C01816=1163.535,366.702,-80.590,-176.202,9.029,148.717
C01817=1163.539,366.455,-80.555,-176.204,9.026,148.716
C01818=1163.543,366.207,-80.520,-176.206,9.021,148.716
C01819=1163.547,365.925,-80.480,-176.209,9.017,148.716
C01820=1163.552,365.642,-80.440,-176.211,9.012,148.715
C01821=1163.557,365.360,-80.400,-176.214,9.008,148.715
C01822=1163.561,365.077,-80.360,-176.217,9.004,148.714
C01823=1163.565,364.830,-80.326,-176.219,9.000,148.714
C01824=1163.569,364.582,-80.290,-176.221,8.996,148.713
C01825=1163.573,364.334,-80.255,-176.223,8.993,148.713
C01826=1163.577,364.087,-80.220,-176.226,8.988,148.713
C01827=1163.581,363.840,-80.186,-176.228,8.985,148.712
C01828=1163.585,363.592,-80.152,-176.230,8.980,148.712
C01829=1163.589,363.345,-80.116,-176.233,8.977,148.712
C01830=1163.593,363.097,-80.081,-176.235,8.974,148.711
C01831=1163.597,362.849,-80.047,-176.237,8.969,148.711
C01832=1163.600,362.602,-80.012,-176.239,8.966,148.711
C01833=1163.605,362.355,-79.977,-176.242,8.962,148.710
C01834=1163.609,362.106,-79.942,-176.244,8.958,148.710
C01835=1163.612,361.860,-79.908,-176.247,8.954,148.710
C01836=1163.616,361.612,-79.873,-176.249,8.950,148.709
C01837=1163.621,361.364,-79.839,-176.252,8.946,148.709
C01838=1163.625,361.116,-79.804,-176.254,8.943,148.709
C01839=1163.628,360.870,-79.769,-176.256,8.939,148.708
C01840=1163.632,360.622,-79.734,-176.259,8.935,148.708
C01841=1163.637,360.374,-79.700,-176.261,8.932,148.708
C01842=1163.640,360.126,-79.666,-176.263,8.928,148.707
C01843=1163.645,359.879,-79.631,-176.265,8.924,148.707
C01844=1163.649,359.631,-79.596,-176.268,8.920,148.707
C01845=1163.652,359.384,-79.562,-176.270,8.917,148.706
C01846=1163.656,359.136,-79.527,-176.273,8.912,148.706
C01847=1163.661,358.889,-79.492,-176.275,8.909,148.706
C01848=1163.664,358.641,-79.458,-176.278,8.905,148.706
C01849=1163.669,358.394,-79.424,-176.280,8.901,148.705
C01850=1163.673,358.145,-79.389,-176.282,8.898,148.705
C01851=1163.676,357.898,-79.355,-176.285,8.894,148.705
C01852=1163.680,357.650,-79.320,-176.287,8.890,148.704
C01853=1163.684,357.403,-79.286,-176.290,8.886,148.704
C01854=1163.688,357.155,-79.251,-176.292,8.883,148.704
C01855=1163.692,356.908,-79.218,-176.294,8.880,148.704
C01856=1163.696,356.660,-79.183,-176.297,8.875,148.703
C01857=1163.701,356.412,-79.148,-176.299,8.872,148.703
C01858=1163.704,356.165,-79.114,-176.302,8.868,148.703
C01859=1163.708,355.917,-79.080,-176.304,8.864,148.702
C01860=1163.712,355.670,-79.046,-176.306,8.861,148.702
C01861=1163.716,355.422,-79.011,-176.309,8.857,148.702
C01862=1163.720,355.175,-78.977,-176.311,8.853,148.701
C01863=1163.725,354.927,-78.943,-176.314,8.849,148.701
C01864=1163.728,354.679,-78.909,-176.316,8.846,148.701
C01865=1163.733,354.432,-78.875,-176.318,8.842,148.701
C01866=1163.736,354.184,-78.840,-176.321,8.838,148.700
C01867=1163.740,353.936,-78.806,-176.324,8.835,148.700
C01868=1163.744,353.689,-78.772,-176.326,8.831,148.700
C01869=1163.748,353.441,-78.737,-176.328,8.827,148.699
C01870=1163.752,353.193,-78.704,-176.331,8.824,148.699
C01871=1163.756,352.946,-78.670,-176.334,8.820,148.699
C01872=1163.760,352.698,-78.635,-176.335,8.816,148.698
C01873=1163.764,352.451,-78.601,-176.338,8.813,148.698
C01874=1163.769,352.203,-78.568,-176.341,8.809,148.698
C01875=1163.772,351.955,-78.533,-176.343,8.806,148.698
C01876=1163.777,351.708,-78.499,-176.346,8.801,148.698
C01877=1163.781,351.460,-78.466,-176.348,8.798,148.697
C01878=1163.784,351.212,-78.432,-176.350,8.795,148.697
C01879=1163.789,350.965,-78.397,-176.353,8.790,148.697
C01880=1163.793,350.717,-78.364,-176.355,8.787,148.696
C01881=1163.796,350.469,-78.330,-176.357,8.784,148.696
C01882=1163.801,350.222,-78.295,-176.360,8.780,148.696
C01883=1163.805,349.974,-78.262,-176.363,8.776,148.696
C01884=1163.809,349.727,-78.228,-176.365,8.773,148.696
C01885=1163.813,349.478,-78.194,-176.367,8.769,148.695
C01886=1163.817,349.231,-78.160,-176.370,8.765,148.695
C01887=1163.821,348.983,-78.127,-176.372,8.762,148.695
C01888=1163.825,348.736,-78.093,-176.375,8.758,148.694
C01889=1163.829,348.488,-78.059,-176.377,8.755,148.694
C01890=1163.833,348.240,-78.025,-176.379,8.752,148.694
C01891=1163.837,347.993,-77.992,-176.382,8.747,148.694
C01892=1163.841,347.745,-77.958,-176.384,8.744,148.693
C01893=1163.845,347.497,-77.924,-176.387,8.741,148.693
C01894=1163.849,347.250,-77.890,-176.389,8.736,148.693
C01895=1163.853,347.002,-77.857,-176.391,8.733,148.693
C01896=1163.858,346.755,-77.823,-176.394,8.730,148.692
C01897=1163.862,346.507,-77.789,-176.397,8.726,148.692
C01898=1163.865,346.258,-77.756,-176.399,8.722,148.692
C01899=1163.869,346.011,-77.722,-176.401,8.719,148.692
C01900=1163.873,345.764,-77.689,-176.404,8.715,148.691
C01901=1163.878,345.516,-77.655,-176.406,8.712,148.691
C01902=1163.882,345.268,-77.621,-176.409,8.708,148.691
C01903=1163.885,345.020,-77.588,-176.412,8.704,148.691
C01904=1163.890,344.772,-77.555,-176.414,8.701,148.691
C01905=1163.893,344.525,-77.521,-176.416,8.698,148.690
C01906=1163.898,344.277,-77.488,-176.419,8.694,148.690
C01907=1163.902,344.029,-77.454,-176.421,8.690,148.690
C01908=1163.907,343.782,-77.421,-176.424,8.687,148.690
C01909=1163.910,343.534,-77.386,-176.426,8.684,148.689
C01910=1163.914,343.286,-77.353,-176.429,8.680,148.689
C01911=1163.918,343.038,-77.320,-176.431,8.676,148.689
C01912=1163.922,342.791,-77.287,-176.433,8.673,148.689
C01913=1163.926,342.543,-77.254,-176.436,8.669,148.688
C01914=1163.930,342.296,-77.220,-176.439,8.666,148.688
C01915=1163.934,342.048,-77.187,-176.441,8.662,148.688
C01916=1163.938,341.800,-77.154,-176.444,8.658,148.688
C01917=1163.943,341.553,-77.120,-176.446,8.655,148.688
C01918=1163.947,341.304,-77.086,-176.448,8.652,148.687
C01919=1163.951,341.056,-77.053,-176.451,8.648,148.687
C01920=1163.955,340.808,-77.020,-176.454,8.644,148.687
C01921=1163.959,340.561,-76.987,-176.456,8.641,148.687
C01922=1163.963,340.313,-76.954,-176.458,8.638,148.687
C01923=1163.968,340.033,-76.916,-176.461,8.634,148.686
C01924=1163.973,339.754,-76.879,-176.464,8.629,148.686
C01925=1163.977,339.474,-76.841,-176.467,8.625,148.686
C01926=1163.981,339.195,-76.804,-176.470,8.621,148.686
C01927=1163.985,338.947,-76.771,-176.472,8.618,148.685
C01928=1163.989,338.700,-76.738,-176.474,8.615,148.685
C01929=1163.993,338.452,-76.705,-176.477,8.612,148.685
C01930=1163.998,338.204,-76.672,-176.480,8.608,148.685
C01931=1164.002,337.956,-76.638,-176.482,8.604,148.685
C01932=1164.006,337.709,-76.605,-176.484,8.601,148.684
C01933=1164.010,337.461,-76.572,-176.487,8.598,148.684
C01934=1164.014,337.213,-76.540,-176.490,8.594,148.684
C01935=1164.019,336.965,-76.507,-176.492,8.590,148.684
C01936=1164.022,336.717,-76.474,-176.494,8.587,148.684
C01937=1164.026,336.470,-76.441,-176.496,8.584,148.683
C01938=1164.030,336.222,-76.408,-176.499,8.580,148.683
C01939=1164.034,335.974,-76.374,-176.502,8.577,148.683
C01940=1164.039,335.726,-76.342,-176.504,8.573,148.683
C01941=1164.043,335.478,-76.309,-176.507,8.570,148.683
C01942=1164.046,335.231,-76.276,-176.510,8.566,148.682
C01943=1164.051,334.983,-76.243,-176.512,8.563,148.682
C01944=1164.055,334.735,-76.211,-176.514,8.559,148.682
C01945=1164.059,334.487,-76.178,-176.516,8.556,148.682
C01946=1164.063,334.239,-76.144,-176.520,8.552,148.682
C01947=1164.067,333.991,-76.113,-176.522,8.549,148.682
C01948=1164.071,333.743,-76.079,-176.524,8.546,148.681
C01949=1164.075,333.496,-76.046,-176.527,8.542,148.681
C01950=1164.080,333.247,-76.014,-176.529,8.538,148.681
C01951=1164.083,333.000,-75.981,-176.532,8.535,148.681
C01952=1164.088,332.753,-75.948,-176.535,8.532,148.681
C01953=1164.092,332.505,-75.916,-176.537,8.529,148.681
C01954=1164.096,332.257,-75.883,-176.539,8.525,148.680
C01955=1164.100,332.009,-75.850,-176.542,8.521,148.680
C01956=1164.104,331.761,-75.818,-176.544,8.518,148.680
C01957=1164.108,331.513,-75.785,-176.547,8.515,148.680
C01958=1164.112,331.265,-75.753,-176.549,8.512,148.680
C01959=1164.116,331.018,-75.720,-176.552,8.508,148.679
C01960=1164.121,330.769,-75.687,-176.554,8.504,148.679
C01961=1164.125,330.522,-75.655,-176.557,8.501,148.679
C01962=1164.129,330.274,-75.623,-176.559,8.498,148.679
C01963=1164.133,330.026,-75.589,-176.562,8.495,148.679
C01964=1164.137,329.778,-75.558,-176.565,8.491,148.679
C01965=1164.141,329.531,-75.524,-176.567,8.487,148.678
C01966=1164.145,329.283,-75.493,-176.569,8.484,148.678
C01967=1164.149,329.034,-75.460,-176.572,8.481,148.678
C01968=1164.154,328.787,-75.427,-176.574,8.478,148.678
C01969=1164.158,328.539,-75.396,-176.577,8.474,148.678
C01970=1164.162,328.291,-75.362,-176.579,8.470,148.678
C01971=1164.166,328.043,-75.331,-176.582,8.467,148.678
C01972=1164.170,327.795,-75.298,-176.584,8.464,148.677
C01973=1164.174,327.548,-75.266,-176.587,8.461,148.677
C01974=1164.178,327.300,-75.233,-176.590,8.457,148.677
C01975=1164.182,327.052,-75.202,-176.592,8.454,148.677
C01976=1164.186,326.804,-75.168,-176.595,8.451,148.677
C01977=1164.190,326.556,-75.137,-176.597,8.447,148.677
C01978=1164.195,326.309,-75.105,-176.599,8.444,148.676
C01979=1164.199,326.060,-75.073,-176.603,8.440,148.676
C01980=1164.203,325.813,-75.040,-176.605,8.437,148.676
C01981=1164.207,325.565,-75.008,-176.607,8.434,148.676
C01982=1164.211,325.316,-74.975,-176.609,8.430,148.676
C01983=1164.215,325.069,-74.944,-176.612,8.427,148.676
C01984=1164.220,324.821,-74.911,-176.615,8.423,148.675
C01985=1164.223,324.573,-74.879,-176.617,8.420,148.675
C01986=1164.228,324.325,-74.846,-176.620,8.417,148.675
C01987=1164.232,324.078,-74.815,-176.622,8.414,148.675
C01988=1164.236,323.830,-74.783,-176.625,8.410,148.675
C01989=1164.240,323.581,-74.751,-176.627,8.407,148.675
C01990=1164.244,323.333,-74.719,-176.630,8.403,148.675
C01991=1164.249,323.085,-74.687,-176.633,8.400,148.674
C01992=1164.253,322.837,-74.655,-176.635,8.397,148.674
C01993=1164.256,322.589,-74.623,-176.638,8.394,148.674
C01994=1164.261,322.342,-74.591,-176.640,8.390,148.674
C01995=1164.265,322.094,-74.559,-176.642,8.387,148.674
C01996=1164.268,321.846,-74.526,-176.646,8.383,148.674
C01997=1164.273,321.599,-74.494,-176.648,8.380,148.674
C01998=1164.277,321.351,-74.463,-176.650,8.377,148.673
C01999=1164.281,321.102,-74.431,-176.653,8.374,148.673
C02000=1164.286,320.854,-74.399,-176.655,8.370,148.673
C02001=1164.290,320.606,-74.368,-176.657,8.367,148.673
C02002=1164.294,320.358,-74.336,-176.661,8.363,148.673
C02003=1164.298,320.111,-74.304,-176.663,8.360,148.673
C02004=1164.302,319.863,-74.272,-176.665,8.357,148.673
C02005=1164.306,319.615,-74.240,-176.668,8.354,148.673
C02006=1164.310,319.367,-74.208,-176.670,8.351,148.672
C02007=1164.314,319.119,-74.177,-176.673,8.348,148.672
C02008=1164.319,318.871,-74.144,-176.675,8.344,148.672
C02009=1164.323,318.623,-74.113,-176.678,8.340,148.672
C02010=1164.327,318.375,-74.082,-176.681,8.337,148.672
C02011=1164.331,318.127,-74.050,-176.683,8.334,148.672
C02012=1164.336,317.879,-74.018,-176.686,8.331,148.672
C02013=1164.339,317.631,-73.986,-176.688,8.328,148.672
C02014=1164.344,317.383,-73.955,-176.691,8.324,148.671
C02015=1164.348,317.135,-73.923,-176.693,8.321,148.672
C02016=1164.351,316.887,-73.891,-176.696,8.317,148.671
C02017=1164.356,316.640,-73.860,-176.699,8.314,148.671
C02018=1164.360,316.391,-73.828,-176.701,8.311,148.671
C02019=1164.365,316.143,-73.797,-176.704,8.308,148.671
C02020=1164.368,315.895,-73.765,-176.706,8.305,148.671
C02021=1164.373,315.647,-73.734,-176.709,8.301,148.671
C02022=1164.377,315.399,-73.702,-176.711,8.298,148.671
C02023=1164.380,315.151,-73.670,-176.714,8.295,148.671
C02024=1164.385,314.903,-73.640,-176.717,8.291,148.670
C02025=1164.389,314.655,-73.608,-176.719,8.288,148.670
C02026=1164.393,314.408,-73.576,-176.722,8.285,148.670
C02027=1164.398,314.131,-73.542,-176.724,8.282,148.670
C02028=1164.403,313.853,-73.506,-176.727,8.278,148.670
C02029=1164.407,313.576,-73.471,-176.731,8.274,148.670
C02030=1164.412,313.299,-73.436,-176.733,8.271,148.670
C02031=1164.416,313.051,-73.405,-176.736,8.268,148.670
C02032=1164.421,312.803,-73.373,-176.738,8.264,148.670
C02033=1164.425,312.555,-73.342,-176.741,8.260,148.669
C02034=1164.429,312.307,-73.310,-176.744,8.257,148.669
C02035=1164.433,312.059,-73.279,-176.746,8.254,148.669
C02036=1164.437,311.811,-73.248,-176.749,8.251,148.669
C02037=1164.441,311.563,-73.217,-176.751,8.248,148.669
C02038=1164.446,311.315,-73.185,-176.754,8.245,148.669
C02039=1164.450,311.067,-73.154,-176.756,8.241,148.669
C02040=1164.454,310.819,-73.123,-176.759,8.239,148.669
C02041=1164.458,310.571,-73.091,-176.761,8.235,148.669
C02042=1164.463,310.323,-73.061,-176.764,8.231,148.669
C02043=1164.467,310.075,-73.030,-176.767,8.228,148.668
C02044=1164.470,309.827,-72.999,-176.769,8.225,148.668
C02045=1164.475,309.579,-72.968,-176.772,8.222,148.668
C02046=1164.479,309.330,-72.937,-176.774,8.219,148.668
C02047=1164.483,309.083,-72.905,-176.777,8.216,148.668
C02048=1164.487,308.834,-72.874,-176.779,8.213,148.668
C02049=1164.492,308.587,-72.843,-176.782,8.209,148.668
C02050=1164.496,308.339,-72.812,-176.784,8.206,148.668
C02051=1164.500,308.091,-72.781,-176.787,8.203,148.668
C02052=1164.505,307.843,-72.750,-176.789,8.200,148.668
C02053=1164.508,307.594,-72.720,-176.792,8.196,148.668
C02054=1164.512,307.347,-72.688,-176.795,8.193,148.668
C02055=1164.517,307.099,-72.657,-176.797,8.190,148.667
C02056=1164.521,306.850,-72.626,-176.800,8.187,148.667
C02057=1164.526,306.602,-72.595,-176.802,8.184,148.667
C02058=1164.530,306.354,-72.565,-176.805,8.181,148.667
C02059=1164.533,306.106,-72.534,-176.807,8.177,148.667
C02060=1164.538,305.859,-72.503,-176.810,8.174,148.667
C02061=1164.542,305.611,-72.472,-176.812,8.171,148.667
C02062=1164.546,305.362,-72.441,-176.815,8.168,148.667
C02063=1164.551,305.114,-72.410,-176.818,8.165,148.667
C02064=1164.555,304.866,-72.380,-176.820,8.162,148.667
C02065=1164.559,304.618,-72.349,-176.823,8.158,148.667
C02066=1164.563,304.370,-72.318,-176.825,8.155,148.667
C02067=1164.568,304.122,-72.287,-176.828,8.151,148.666
C02068=1164.571,303.874,-72.257,-176.831,8.148,148.666
C02069=1164.576,303.626,-72.226,-176.834,8.145,148.666
C02070=1164.581,303.378,-72.195,-176.836,8.142,148.666
C02071=1164.584,303.130,-72.165,-176.839,8.139,148.666
C02072=1164.588,302.881,-72.134,-176.841,8.136,148.666
C02073=1164.593,302.633,-72.103,-176.844,8.133,148.666
C02074=1164.597,302.386,-72.073,-176.846,8.130,148.666
C02075=1164.601,302.137,-72.042,-176.849,8.127,148.666
C02076=1164.606,301.889,-72.011,-176.852,8.124,148.666
C02077=1164.609,301.641,-71.981,-176.854,8.120,148.666
C02078=1164.614,301.393,-71.950,-176.857,8.117,148.666
C02079=1164.618,301.144,-71.920,-176.859,8.114,148.666
C02080=1164.622,300.897,-71.889,-176.862,8.111,148.666
C02081=1164.627,300.649,-71.859,-176.864,8.108,148.665
C02082=1164.631,300.401,-71.828,-176.867,8.105,148.665
C02083=1164.635,300.153,-71.798,-176.869,8.102,148.666
C02084=1164.639,299.904,-71.767,-176.872,8.099,148.665
C02085=1164.644,299.656,-71.737,-176.874,8.096,148.665
C02086=1164.648,299.408,-71.706,-176.877,8.092,148.665
C02087=1164.652,299.160,-71.676,-176.880,8.089,148.665
C02088=1164.656,298.912,-71.645,-176.883,8.086,148.665
C02089=1164.660,298.664,-71.616,-176.885,8.082,148.665
C02090=1164.665,298.416,-71.585,-176.888,8.079,148.665
C02091=1164.669,298.168,-71.555,-176.891,8.076,148.665
C02092=1164.673,297.920,-71.524,-176.893,8.073,148.665
C02093=1164.678,297.672,-71.494,-176.896,8.070,148.665
C02094=1164.682,297.423,-71.463,-176.898,8.067,148.665
C02095=1164.685,297.175,-71.433,-176.901,8.064,148.665
C02096=1164.690,296.927,-71.403,-176.903,8.061,148.665
C02097=1164.694,296.679,-71.373,-176.906,8.058,148.665
C02098=1164.699,296.431,-71.343,-176.908,8.055,148.665
C02099=1164.703,296.183,-71.313,-176.911,8.052,148.665
C02100=1164.707,295.934,-71.282,-176.914,8.048,148.665
C02101=1164.711,295.686,-71.252,-176.916,8.045,148.665
C02102=1164.716,295.438,-71.221,-176.919,8.042,148.664
C02103=1164.720,295.190,-71.192,-176.921,8.039,148.664
C02104=1164.724,294.942,-71.162,-176.924,8.036,148.664
C02105=1164.729,294.694,-71.132,-176.926,8.033,148.664
C02106=1164.733,294.446,-71.102,-176.929,8.030,148.664
C02107=1164.737,294.198,-71.072,-176.932,8.027,148.664
C02108=1164.741,293.949,-71.041,-176.934,8.024,148.664
C02109=1164.745,293.701,-71.012,-176.937,8.021,148.664
C02110=1164.750,293.453,-70.981,-176.940,8.018,148.664
C02111=1164.754,293.204,-70.951,-176.942,8.015,148.664
C02112=1164.758,292.957,-70.921,-176.945,8.012,148.664
C02113=1164.763,292.708,-70.891,-176.947,8.009,148.664
C02114=1164.766,292.461,-70.861,-176.950,8.006,148.664
C02115=1164.771,292.212,-70.831,-176.952,8.002,148.664
C02116=1164.775,291.964,-70.802,-176.955,7.999,148.664
C02117=1164.779,291.716,-70.771,-176.958,7.996,148.664
C02118=1164.784,291.468,-70.742,-176.960,7.993,148.664
C02119=1164.788,291.220,-70.712,-176.963,7.990,148.664
C02120=1164.792,290.972,-70.682,-176.966,7.987,148.664
C02121=1164.797,290.723,-70.652,-176.968,7.984,148.664
C02122=1164.801,290.475,-70.623,-176.971,7.981,148.664
C02123=1164.805,290.227,-70.592,-176.974,7.978,148.664
C02124=1164.810,289.979,-70.562,-176.976,7.975,148.664
C02125=1164.813,289.730,-70.533,-176.979,7.972,148.664
C02126=1164.817,289.482,-70.503,-176.981,7.969,148.664
C02127=1164.821,289.234,-70.473,-176.984,7.966,148.664
C02128=1164.825,288.986,-70.444,-176.986,7.962,148.664
C02129=1164.831,288.738,-70.414,-176.989,7.960,148.664
C02130=1164.835,288.490,-70.384,-176.992,7.957,148.664
C02131=1164.840,288.215,-70.351,-176.995,7.954,148.664
C02132=1164.844,287.940,-70.319,-176.998,7.949,148.663
C02133=1164.849,287.665,-70.286,-177.000,7.947,148.663
C02134=1164.854,287.390,-70.253,-177.004,7.943,148.663
C02135=1164.858,287.141,-70.224,-177.006,7.940,148.663
C02136=1164.862,286.893,-70.194,-177.009,7.938,148.664
C02137=1164.867,286.645,-70.163,-177.011,7.934,148.663
C02138=1164.871,286.397,-70.134,-177.014,7.931,148.663
C02139=1164.875,286.149,-70.105,-177.016,7.928,148.663
C02140=1164.879,285.900,-70.075,-177.019,7.925,148.664
C02141=1164.883,285.652,-70.046,-177.021,7.922,148.663
C02142=1164.887,285.404,-70.016,-177.024,7.919,148.663
C02143=1164.892,285.155,-69.987,-177.027,7.916,148.663
C02144=1164.896,284.908,-69.958,-177.030,7.913,148.663
C02145=1164.901,284.660,-69.928,-177.032,7.910,148.663
C02146=1164.905,284.411,-69.899,-177.035,7.907,148.663
C02147=1164.909,284.163,-69.869,-177.037,7.904,148.663
C02148=1164.913,283.915,-69.840,-177.040,7.901,148.663
C02149=1164.917,283.667,-69.810,-177.042,7.898,148.663
C02150=1164.922,283.418,-69.782,-177.045,7.895,148.663
C02151=1164.926,283.169,-69.752,-177.048,7.892,148.663
C02152=1164.931,282.922,-69.723,-177.051,7.889,148.663
C02153=1164.935,282.674,-69.694,-177.053,7.886,148.663
C02154=1164.939,282.425,-69.664,-177.056,7.883,148.663
C02155=1164.943,282.177,-69.635,-177.059,7.880,148.663
C02156=1164.947,281.929,-69.605,-177.061,7.877,148.663
C02157=1164.952,281.680,-69.577,-177.064,7.874,148.663
C02158=1164.956,281.432,-69.547,-177.066,7.872,148.663
C02159=1164.961,281.184,-69.518,-177.068,7.868,148.663
C02160=1164.965,280.936,-69.489,-177.071,7.865,148.663
C02161=1164.969,280.688,-69.459,-177.074,7.862,148.663
C02162=1164.974,280.439,-69.430,-177.077,7.859,148.663
C02163=1164.978,280.190,-69.401,-177.079,7.856,148.663
C02164=1164.983,279.943,-69.372,-177.082,7.853,148.663
C02165=1164.987,279.695,-69.342,-177.085,7.850,148.663
C02166=1164.991,279.446,-69.314,-177.087,7.847,148.663
C02167=1164.995,279.198,-69.285,-177.090,7.844,148.663
C02168=1164.999,278.949,-69.255,-177.093,7.841,148.663
C02169=1165.004,278.701,-69.227,-177.096,7.838,148.663
C02170=1165.008,278.453,-69.198,-177.098,7.835,148.663
C02171=1165.013,278.205,-69.168,-177.101,7.832,148.663
C02172=1165.016,277.956,-69.140,-177.103,7.829,148.663
C02173=1165.021,277.709,-69.111,-177.106,7.827,148.663
C02174=1165.026,277.460,-69.082,-177.108,7.824,148.664
C02175=1165.030,277.211,-69.053,-177.111,7.821,148.664
C02176=1165.034,276.963,-69.023,-177.114,7.818,148.664
C02177=1165.038,276.715,-68.995,-177.116,7.815,148.663
C02178=1165.042,276.467,-68.966,-177.119,7.812,148.663
C02179=1165.047,276.218,-68.937,-177.122,7.809,148.664
C02180=1165.051,275.970,-68.908,-177.124,7.806,148.664
C02181=1165.055,275.722,-68.880,-177.127,7.803,148.664
C02182=1165.060,275.474,-68.851,-177.130,7.800,148.664
C02183=1165.064,275.225,-68.822,-177.133,7.797,148.664
C02184=1165.068,274.977,-68.793,-177.134,7.795,148.664
C02185=1165.073,274.729,-68.765,-177.137,7.792,148.664
C02186=1165.077,274.480,-68.735,-177.140,7.789,148.664
C02187=1165.081,274.232,-68.706,-177.143,7.786,148.664
C02188=1165.086,273.984,-68.679,-177.145,7.783,148.664
C02189=1165.090,273.735,-68.649,-177.148,7.780,148.664
C02190=1165.094,273.486,-68.620,-177.151,7.777,148.664
C02191=1165.099,273.239,-68.593,-177.154,7.774,148.664
C02192=1165.103,272.990,-68.563,-177.156,7.771,148.664
C02193=1165.107,272.742,-68.535,-177.158,7.768,148.664
C02194=1165.111,272.494,-68.506,-177.161,7.765,148.664
C02195=1165.116,272.245,-68.477,-177.164,7.763,148.664
C02196=1165.120,271.997,-68.449,-177.166,7.760,148.664
C02197=1165.125,271.749,-68.421,-177.169,7.757,148.664
C02198=1165.129,271.500,-68.391,-177.172,7.754,148.664
C02199=1165.133,271.252,-68.363,-177.175,7.751,148.664
C02200=1165.138,271.004,-68.335,-177.177,7.748,148.664
C02201=1165.141,270.755,-68.307,-177.180,7.745,148.664
C02202=1165.146,270.507,-68.278,-177.182,7.743,148.664
C02203=1165.150,270.259,-68.249,-177.185,7.740,148.664
C02204=1165.155,270.011,-68.221,-177.188,7.737,148.664
C02205=1165.159,269.762,-68.193,-177.190,7.733,148.664
C02206=1165.163,269.513,-68.164,-177.193,7.730,148.664
C02207=1165.168,269.266,-68.135,-177.196,7.728,148.664
C02208=1165.172,269.017,-68.107,-177.198,7.725,148.664
C02209=1165.177,268.769,-68.079,-177.201,7.722,148.664
C02210=1165.181,268.520,-68.050,-177.203,7.719,148.665
C02211=1165.186,268.272,-68.022,-177.206,7.716,148.665
C02212=1165.190,268.023,-67.994,-177.209,7.714,148.665
C02213=1165.194,267.776,-67.966,-177.212,7.711,148.665
C02214=1165.198,267.527,-67.937,-177.214,7.708,148.665
C02215=1165.202,267.278,-67.909,-177.217,7.705,148.665
C02216=1165.207,267.030,-67.881,-177.220,7.702,148.665
C02217=1165.211,266.781,-67.853,-177.222,7.700,148.665
C02218=1165.216,266.533,-67.824,-177.225,7.697,148.665
C02219=1165.220,266.285,-67.796,-177.228,7.694,148.665
C02220=1165.225,266.036,-67.768,-177.230,7.691,148.665
C02221=1165.229,265.788,-67.740,-177.233,7.688,148.665
C02222=1165.233,265.540,-67.712,-177.236,7.685,148.665
C02223=1165.237,265.291,-67.683,-177.238,7.683,148.665
C02224=1165.242,265.043,-67.655,-177.241,7.680,148.665
C02225=1165.246,264.794,-67.627,-177.243,7.677,148.665
C02226=1165.251,264.546,-67.599,-177.246,7.674,148.665
C02227=1165.254,264.298,-67.571,-177.249,7.671,148.666
C02228=1165.260,264.050,-67.542,-177.252,7.668,148.666
C02229=1165.264,263.802,-67.515,-177.255,7.665,148.666
C02230=1165.268,263.553,-67.486,-177.257,7.663,148.666
C02231=1165.273,263.304,-67.459,-177.259,7.660,148.666
C02232=1165.277,263.056,-67.431,-177.262,7.657,148.666
C02233=1165.281,262.808,-67.403,-177.265,7.654,148.666
C02234=1165.285,262.559,-67.375,-177.268,7.651,148.666
C02235=1165.290,262.286,-67.343,-177.270,7.648,148.666
C02236=1165.296,262.013,-67.313,-177.273,7.645,148.666
C02237=1165.300,261.740,-67.282,-177.276,7.642,148.666
C02238=1165.305,261.466,-67.252,-177.279,7.638,148.666
C02239=1165.309,261.219,-67.224,-177.282,7.636,148.666
C02240=1165.313,260.970,-67.196,-177.284,7.633,148.666
C02241=1165.318,260.722,-67.169,-177.287,7.630,148.666
C02242=1165.322,260.473,-67.140,-177.290,7.627,148.666
C02243=1165.326,260.225,-67.112,-177.293,7.624,148.666
C02244=1165.331,259.976,-67.085,-177.295,7.622,148.667
C02245=1165.335,259.728,-67.057,-177.297,7.619,148.667
C02246=1165.339,259.480,-67.029,-177.300,7.616,148.667
C02247=1165.345,259.231,-67.002,-177.303,7.613,148.667
C02248=1165.348,258.982,-66.973,-177.306,7.611,148.667
C02249=1165.353,258.735,-66.946,-177.308,7.609,148.667
C02250=1165.357,258.485,-66.918,-177.311,7.606,148.667
C02251=1165.361,258.237,-66.890,-177.314,7.603,148.667
C02252=1165.366,257.989,-66.863,-177.317,7.600,148.667
C02253=1165.370,257.740,-66.835,-177.319,7.597,148.667
C02254=1165.375,257.492,-66.808,-177.322,7.595,148.667
C02255=1165.379,257.244,-66.780,-177.324,7.592,148.667
C02256=1165.383,256.995,-66.752,-177.327,7.589,148.668
C02257=1165.388,256.747,-66.725,-177.330,7.586,148.668
C02258=1165.392,256.498,-66.698,-177.333,7.583,148.668
C02259=1165.397,256.250,-66.670,-177.335,7.581,148.668
C02260=1165.401,256.001,-66.642,-177.338,7.578,148.668
C02261=1165.405,255.753,-66.615,-177.340,7.575,148.668
C02262=1165.410,255.505,-66.588,-177.344,7.572,148.668
C02263=1165.413,255.256,-66.559,-177.346,7.569,148.668
C02264=1165.418,255.008,-66.532,-177.349,7.567,148.668
C02265=1165.423,254.759,-66.505,-177.351,7.564,148.668
C02266=1165.427,254.511,-66.478,-177.354,7.561,148.668
C02267=1165.431,254.262,-66.450,-177.357,7.558,148.668
C02268=1165.436,254.014,-66.422,-177.359,7.556,148.669
C02269=1165.440,253.766,-66.395,-177.362,7.553,148.669
C02270=1165.445,253.517,-66.368,-177.364,7.550,148.669
C02271=1165.449,253.269,-66.340,-177.368,7.547,148.669
C02272=1165.453,253.020,-66.313,-177.370,7.545,148.669
C02273=1165.458,252.772,-66.286,-177.373,7.542,148.669
C02274=1165.463,252.523,-66.259,-177.375,7.539,148.669
C02275=1165.466,252.275,-66.231,-177.378,7.536,148.669
C02276=1165.471,252.026,-66.204,-177.381,7.534,148.669
C02277=1165.476,251.778,-66.177,-177.383,7.531,148.669
C02278=1165.480,251.529,-66.150,-177.386,7.528,148.670
C02279=1165.485,251.281,-66.122,-177.389,7.526,148.670
C02280=1165.489,251.032,-66.094,-177.392,7.523,148.670
C02281=1165.493,250.784,-66.068,-177.394,7.521,148.670
C02282=1165.497,250.535,-66.041,-177.397,7.518,148.670
C02283=1165.502,250.287,-66.014,-177.400,7.515,148.670
C02284=1165.506,250.039,-65.986,-177.402,7.512,148.670
C02285=1165.510,249.790,-65.959,-177.405,7.510,148.670
C02286=1165.515,249.541,-65.931,-177.408,7.507,148.671
C02287=1165.520,249.293,-65.904,-177.411,7.504,148.671
C02288=1165.524,249.045,-65.878,-177.413,7.502,148.671
C02289=1165.528,248.796,-65.851,-177.415,7.499,148.671
C02290=1165.533,248.548,-65.824,-177.418,7.496,148.671
C02291=1165.537,248.298,-65.796,-177.421,7.493,148.671
C02292=1165.542,248.050,-65.769,-177.424,7.491,148.671
C02293=1165.546,247.802,-65.743,-177.426,7.488,148.671
C02294=1165.550,247.553,-65.716,-177.429,7.485,148.671
C02295=1165.555,247.305,-65.689,-177.432,7.482,148.671
C02296=1165.560,247.056,-65.662,-177.434,7.480,148.672
C02297=1165.564,246.808,-65.635,-177.437,7.477,148.672
C02298=1165.568,246.560,-65.608,-177.440,7.475,148.672
C02299=1165.573,246.311,-65.581,-177.442,7.473,148.672
C02300=1165.577,246.062,-65.554,-177.445,7.470,148.672
C02301=1165.581,245.814,-65.527,-177.448,7.467,148.672
C02302=1165.585,245.565,-65.500,-177.451,7.464,148.672
C02303=1165.590,245.317,-65.473,-177.453,7.462,148.672
C02304=1165.595,245.068,-65.446,-177.456,7.459,148.673
C02305=1165.599,244.820,-65.420,-177.459,7.456,148.673
C02306=1165.603,244.572,-65.392,-177.461,7.454,148.673
C02307=1165.608,244.322,-65.366,-177.464,7.451,148.673
C02308=1165.612,244.074,-65.340,-177.467,7.448,148.673
C02309=1165.617,243.826,-65.313,-177.470,7.445,148.673
C02310=1165.621,243.577,-65.286,-177.472,7.443,148.673
C02311=1165.625,243.329,-65.259,-177.475,7.440,148.673
C02312=1165.630,243.081,-65.232,-177.478,7.438,148.674
C02313=1165.634,242.832,-65.206,-177.480,7.436,148.674
C02314=1165.639,242.583,-65.179,-177.483,7.433,148.674
C02315=1165.644,242.335,-65.152,-177.486,7.430,148.674
C02316=1165.647,242.087,-65.126,-177.488,7.428,148.674
C02317=1165.652,241.837,-65.099,-177.491,7.425,148.674
C02318=1165.656,241.589,-65.073,-177.494,7.422,148.674
C02319=1165.661,241.341,-65.046,-177.497,7.419,148.674
C02320=1165.666,241.092,-65.019,-177.499,7.417,148.675
C02321=1165.670,240.843,-64.993,-177.502,7.414,148.675
C02322=1165.675,240.595,-64.966,-177.505,7.411,148.675
C02323=1165.679,240.346,-64.940,-177.507,7.409,148.675
C02324=1165.683,240.098,-64.913,-177.510,7.407,148.675
C02325=1165.687,239.849,-64.887,-177.513,7.404,148.675
C02326=1165.692,239.600,-64.860,-177.515,7.402,148.675
C02327=1165.696,239.352,-64.834,-177.518,7.399,148.675
C02328=1165.701,239.103,-64.807,-177.521,7.396,148.676
C02329=1165.705,238.855,-64.781,-177.523,7.394,148.676
C02330=1165.710,238.606,-64.754,-177.526,7.391,148.676
C02331=1165.714,238.358,-64.728,-177.529,7.388,148.676
C02332=1165.719,238.109,-64.701,-177.531,7.386,148.676
C02333=1165.723,237.860,-64.675,-177.534,7.383,148.676
C02334=1165.728,237.612,-64.648,-177.537,7.380,148.676
C02335=1165.732,237.363,-64.623,-177.540,7.378,148.677
C02336=1165.736,237.116,-64.596,-177.542,7.376,148.677
C02337=1165.741,236.866,-64.570,-177.545,7.373,148.677
C02338=1165.745,236.618,-64.544,-177.547,7.370,148.677
C02339=1165.751,236.346,-64.515,-177.551,7.368,148.677
C02340=1165.755,236.075,-64.486,-177.553,7.365,148.677
C02341=1165.760,235.803,-64.458,-177.557,7.362,148.678
C02342=1165.765,235.531,-64.429,-177.559,7.359,148.678
C02343=1165.769,235.282,-64.403,-177.562,7.356,148.678
C02344=1165.774,235.034,-64.376,-177.565,7.355,148.678
C02345=1165.778,234.785,-64.350,-177.568,7.352,148.678
C02346=1165.782,234.536,-64.325,-177.570,7.349,148.678
C02347=1165.787,234.289,-64.298,-177.573,7.347,148.679
C02348=1165.792,234.040,-64.272,-177.576,7.344,148.679
C02349=1165.796,233.791,-64.246,-177.578,7.341,148.679
C02350=1165.801,233.542,-64.219,-177.581,7.339,148.679
C02351=1165.805,233.294,-64.194,-177.584,7.336,148.679
C02352=1165.809,233.045,-64.168,-177.586,7.334,148.679
C02353=1165.814,232.797,-64.142,-177.589,7.332,148.680
C02354=1165.818,232.548,-64.115,-177.592,7.329,148.680
C02355=1165.823,232.299,-64.090,-177.594,7.326,148.680
C02356=1165.827,232.051,-64.064,-177.598,7.324,148.680
C02357=1165.832,231.801,-64.038,-177.600,7.321,148.680
C02358=1165.836,231.554,-64.011,-177.602,7.319,148.680
C02359=1165.841,231.305,-63.986,-177.606,7.316,148.681
C02360=1165.845,231.056,-63.960,-177.608,7.314,148.681
C02361=1165.849,230.808,-63.934,-177.611,7.311,148.681
C02362=1165.854,230.558,-63.908,-177.614,7.308,148.681
C02363=1165.859,230.310,-63.882,-177.616,7.306,148.681
C02364=1165.863,230.062,-63.857,-177.619,7.304,148.682
C02365=1165.867,229.813,-63.830,-177.622,7.302,148.682
C02366=1165.871,229.565,-63.804,-177.624,7.299,148.682
C02367=1165.877,229.316,-63.778,-177.628,7.296,148.682
C02368=1165.881,229.067,-63.753,-177.630,7.294,148.682
C02369=1165.885,228.819,-63.727,-177.632,7.291,148.682
C02370=1165.889,228.570,-63.701,-177.635,7.289,148.683
C02371=1165.894,228.322,-63.676,-177.638,7.286,148.683
C02372=1165.898,228.073,-63.650,-177.641,7.284,148.683
C02373=1165.903,227.824,-63.624,-177.643,7.281,148.683
C02374=1165.908,227.576,-63.599,-177.646,7.279,148.683
C02375=1165.912,227.327,-63.573,-177.649,7.277,148.683
C02376=1165.917,227.078,-63.547,-177.652,7.274,148.684
C02377=1165.921,226.829,-63.521,-177.654,7.272,148.684
C02378=1165.926,226.581,-63.496,-177.657,7.269,148.684
C02379=1165.930,226.332,-63.470,-177.660,7.266,148.684
C02380=1165.934,226.083,-63.444,-177.662,7.264,148.684
C02381=1165.939,225.835,-63.419,-177.665,7.261,148.684
C02382=1165.943,225.587,-63.393,-177.668,7.260,148.685
C02383=1165.948,225.337,-63.368,-177.671,7.257,148.685
C02384=1165.953,225.089,-63.343,-177.673,7.255,148.685
C02385=1165.957,224.840,-63.317,-177.676,7.252,148.685
C02386=1165.961,224.591,-63.291,-177.679,7.249,148.685
C02387=1165.966,224.343,-63.266,-177.681,7.247,148.686
C02388=1165.970,224.095,-63.240,-177.684,7.244,148.686
C02389=1165.975,223.846,-63.215,-177.686,7.242,148.686
C02390=1165.979,223.597,-63.190,-177.690,7.240,148.686
C02391=1165.984,223.348,-63.164,-177.692,7.237,148.686
C02392=1165.989,223.100,-63.138,-177.695,7.235,148.687
C02393=1165.993,222.851,-63.113,-177.697,7.233,148.687
C02394=1165.997,222.602,-63.088,-177.701,7.230,148.687
C02395=1166.002,222.354,-63.062,-177.703,7.227,148.687
C02396=1166.006,222.105,-63.037,-177.705,7.225,148.687
C02397=1166.011,221.857,-63.011,-177.709,7.222,148.688
C02398=1166.016,221.607,-62.986,-177.711,7.220,148.688
C02399=1166.021,221.359,-62.961,-177.714,7.218,148.688
C02400=1166.024,221.111,-62.936,-177.716,7.216,148.688
C02401=1166.029,220.861,-62.911,-177.720,7.213,148.688
C02402=1166.033,220.613,-62.885,-177.722,7.211,148.688
C02403=1166.038,220.364,-62.859,-177.725,7.208,148.689
C02404=1166.043,220.116,-62.835,-177.727,7.206,148.689
C02405=1166.047,219.867,-62.809,-177.730,7.203,148.689
C02406=1166.052,219.618,-62.784,-177.733,7.201,148.689
C02407=1166.056,219.370,-62.759,-177.735,7.198,148.689
C02408=1166.060,219.121,-62.733,-177.738,7.197,148.690
C02409=1166.065,218.872,-62.709,-177.741,7.194,148.690
C02410=1166.069,218.623,-62.683,-177.744,7.192,148.690
C02411=1166.074,218.375,-62.658,-177.746,7.189,148.690
C02412=1166.078,218.126,-62.633,-177.749,7.187,148.691
C02413=1166.083,217.877,-62.609,-177.752,7.184,148.691
C02414=1166.087,217.629,-62.583,-177.754,7.182,148.691
C02415=1166.092,217.380,-62.558,-177.757,7.180,148.691
C02416=1166.096,217.131,-62.532,-177.760,7.178,148.691
C02417=1166.101,216.883,-62.508,-177.763,7.175,148.692
C02418=1166.105,216.634,-62.483,-177.765,7.173,148.692
C02419=1166.110,216.385,-62.458,-177.768,7.170,148.692
C02420=1166.114,216.137,-62.433,-177.771,7.168,148.692
C02421=1166.119,215.888,-62.408,-177.773,7.165,148.692
C02422=1166.123,215.639,-62.383,-177.776,7.164,148.693
C02423=1166.128,215.390,-62.358,-177.779,7.161,148.693
C02424=1166.133,215.142,-62.334,-177.782,7.159,148.693
C02425=1166.137,214.893,-62.308,-177.784,7.156,148.693
C02426=1166.142,214.645,-62.283,-177.787,7.154,148.694
C02427=1166.146,214.395,-62.259,-177.790,7.151,148.694
C02428=1166.151,214.147,-62.233,-177.792,7.149,148.694
C02429=1166.155,213.898,-62.208,-177.795,7.146,148.694
C02430=1166.160,213.649,-62.184,-177.798,7.145,148.694
C02431=1166.164,213.400,-62.159,-177.801,7.142,148.695
C02432=1166.169,213.152,-62.134,-177.803,7.140,148.695
C02433=1166.173,212.904,-62.110,-177.806,7.137,148.695
C02434=1166.178,212.654,-62.085,-177.809,7.135,148.695
C02435=1166.182,212.406,-62.060,-177.812,7.132,148.695
C02436=1166.186,212.157,-62.035,-177.814,7.131,148.696
C02437=1166.192,211.908,-62.010,-177.817,7.128,148.696
C02438=1166.196,211.660,-61.986,-177.820,7.126,148.696
C02439=1166.200,211.410,-61.961,-177.822,7.124,148.697
C02440=1166.205,211.163,-61.936,-177.825,7.121,148.697
C02441=1166.210,210.914,-61.912,-177.828,7.119,148.697
C02442=1166.213,210.665,-61.887,-177.831,7.116,148.697
C02443=1166.219,210.395,-61.860,-177.834,7.114,148.697
C02444=1166.223,210.124,-61.833,-177.836,7.112,148.697
C02445=1166.228,209.853,-61.807,-177.839,7.109,148.698
C02446=1166.233,209.583,-61.780,-177.842,7.106,148.698
C02447=1166.238,209.334,-61.755,-177.845,7.104,148.698
C02448=1166.242,209.085,-61.731,-177.848,7.102,148.699
C02449=1166.248,208.837,-61.706,-177.851,7.100,148.699
C02450=1166.251,208.588,-61.682,-177.853,7.097,148.699
C02451=1166.256,208.339,-61.657,-177.856,7.095,148.699
C02452=1166.261,208.090,-61.633,-177.858,7.093,148.699
C02453=1166.265,207.841,-61.608,-177.861,7.091,148.700
C02454=1166.270,207.593,-61.584,-177.864,7.088,148.700
C02455=1166.275,207.344,-61.559,-177.867,7.086,148.700
C02456=1166.279,207.096,-61.535,-177.869,7.084,148.700
C02457=1166.284,206.846,-61.510,-177.872,7.081,148.701
C02458=1166.288,206.598,-61.486,-177.875,7.079,148.701
C02459=1166.293,206.349,-61.462,-177.877,7.077,148.701
C02460=1166.297,206.100,-61.437,-177.880,7.075,148.701
C02461=1166.302,205.851,-61.413,-177.883,7.072,148.702
C02462=1166.307,205.603,-61.388,-177.886,7.070,148.702
C02463=1166.311,205.354,-61.365,-177.889,7.068,148.702
C02464=1166.315,205.105,-61.340,-177.891,7.065,148.702
C02465=1166.320,204.856,-61.316,-177.894,7.063,148.703
C02466=1166.325,204.607,-61.292,-177.896,7.061,148.703
C02467=1166.330,204.359,-61.267,-177.899,7.059,148.703
C02468=1166.334,204.110,-61.242,-177.902,7.057,148.703
C02469=1166.338,203.861,-61.218,-177.905,7.054,148.704
C02470=1166.343,203.612,-61.195,-177.908,7.052,148.704
C02471=1166.348,203.363,-61.170,-177.910,7.050,148.704
C02472=1166.352,203.115,-61.146,-177.913,7.047,148.704
C02473=1166.356,202.866,-61.122,-177.916,7.046,148.705
C02474=1166.361,202.617,-61.097,-177.919,7.043,148.705
C02475=1166.366,202.368,-61.074,-177.921,7.041,148.705
C02476=1166.370,202.120,-61.050,-177.923,7.039,148.705
C02477=1166.375,201.871,-61.026,-177.927,7.036,148.706
C02478=1166.379,201.621,-61.001,-177.929,7.034,148.706
C02479=1166.384,201.373,-60.977,-177.932,7.032,148.706
C02480=1166.388,201.124,-60.953,-177.935,7.030,148.706
C02481=1166.393,200.876,-60.929,-177.937,7.028,148.707
C02482=1166.398,200.627,-60.905,-177.940,7.025,148.707
C02483=1166.403,200.378,-60.881,-177.943,7.023,148.707
C02484=1166.406,200.129,-60.857,-177.945,7.021,148.707
C02485=1166.411,199.880,-60.833,-177.948,7.019,148.708
C02486=1166.415,199.632,-60.809,-177.951,7.017,148.708
C02487=1166.421,199.382,-60.785,-177.954,7.014,148.708
C02488=1166.425,199.134,-60.761,-177.956,7.012,148.708
C02489=1166.430,198.886,-60.737,-177.959,7.010,148.709
C02490=1166.434,198.637,-60.714,-177.962,7.007,148.709
C02491=1166.438,198.387,-60.689,-177.965,7.006,148.709
C02492=1166.443,198.138,-60.666,-177.967,7.004,148.709
C02493=1166.448,197.890,-60.641,-177.970,7.001,148.710
C02494=1166.453,197.641,-60.618,-177.973,6.999,148.710
C02495=1166.457,197.392,-60.594,-177.975,6.997,148.710
C02496=1166.462,197.143,-60.571,-177.978,6.994,148.711
C02497=1166.466,196.895,-60.546,-177.981,6.993,148.711
C02498=1166.471,196.646,-60.523,-177.984,6.990,148.711
C02499=1166.475,196.397,-60.499,-177.986,6.988,148.711
C02500=1166.480,196.148,-60.476,-177.989,6.986,148.712
C02501=1166.484,195.900,-60.452,-177.992,6.983,148.712
C02502=1166.489,195.650,-60.427,-177.994,6.981,148.712
C02503=1166.494,195.401,-60.403,-177.997,6.980,148.712
C02504=1166.498,195.152,-60.380,-178.000,6.977,148.713
C02505=1166.503,194.903,-60.356,-178.003,6.975,148.713
C02506=1166.507,194.655,-60.332,-178.005,6.973,148.713
C02507=1166.512,194.406,-60.309,-178.008,6.970,148.713
C02508=1166.517,194.157,-60.286,-178.011,6.969,148.714
C02509=1166.521,193.908,-60.262,-178.013,6.967,148.714
C02510=1166.526,193.659,-60.238,-178.016,6.964,148.714
C02511=1166.531,193.410,-60.215,-178.019,6.962,148.715
C02512=1166.535,193.162,-60.191,-178.022,6.960,148.715
C02513=1166.540,192.913,-60.167,-178.025,6.958,148.715
C02514=1166.544,192.664,-60.144,-178.027,6.956,148.715
C02515=1166.549,192.415,-60.120,-178.030,6.954,148.716
C02516=1166.553,192.166,-60.097,-178.033,6.951,148.716
C02517=1166.558,191.917,-60.073,-178.035,6.949,148.716
C02518=1166.563,191.668,-60.050,-178.038,6.947,148.717
C02519=1166.567,191.420,-60.026,-178.040,6.946,148.717
C02520=1166.571,191.171,-60.003,-178.043,6.943,148.717
C02521=1166.576,190.922,-59.980,-178.046,6.941,148.717
C02522=1166.581,190.673,-59.956,-178.049,6.939,148.718
C02523=1166.585,190.424,-59.933,-178.052,6.937,148.718
C02524=1166.590,190.176,-59.909,-178.054,6.934,148.718
C02525=1166.594,189.927,-59.886,-178.057,6.933,148.719
C02526=1166.600,189.678,-59.863,-178.060,6.930,148.719
C02527=1166.604,189.429,-59.839,-178.062,6.928,148.719
C02528=1166.609,189.180,-59.816,-178.065,6.926,148.719
C02529=1166.613,188.932,-59.793,-178.068,6.924,148.720
C02530=1166.618,188.683,-59.770,-178.071,6.922,148.720
C02531=1166.622,188.434,-59.746,-178.073,6.920,148.720
C02532=1166.627,188.185,-59.723,-178.076,6.918,148.721
C02533=1166.632,187.936,-59.699,-178.079,6.915,148.721
C02534=1166.636,187.687,-59.676,-178.081,6.913,148.721
C02535=1166.640,187.438,-59.653,-178.084,6.912,148.721
C02536=1166.645,187.189,-59.630,-178.087,6.909,148.722
C02537=1166.650,186.941,-59.607,-178.090,6.907,148.722
C02538=1166.655,186.692,-59.583,-178.092,6.905,148.722
C02539=1166.660,186.443,-59.560,-178.095,6.903,148.723
C02540=1166.664,186.194,-59.537,-178.098,6.901,148.723
C02541=1166.668,185.945,-59.514,-178.101,6.899,148.723
C02542=1166.673,185.696,-59.490,-178.103,6.897,148.723
C02543=1166.678,185.447,-59.467,-178.105,6.895,148.724
C02544=1166.682,185.198,-59.445,-178.109,6.892,148.724
C02545=1166.687,184.949,-59.422,-178.111,6.891,148.724
C02546=1166.692,184.700,-59.399,-178.114,6.889,148.725
C02547=1166.697,184.431,-59.374,-178.117,6.886,148.725
C02548=1166.702,184.162,-59.348,-178.120,6.884,148.725
C02549=1166.707,183.892,-59.323,-178.123,6.882,148.726
C02550=1166.711,183.623,-59.299,-178.125,6.880,148.726
C02551=1166.716,183.374,-59.276,-178.129,6.877,148.726
C02552=1166.721,183.125,-59.252,-178.131,6.876,148.727
C02553=1166.725,182.875,-59.230,-178.134,6.873,148.727
C02554=1166.730,182.626,-59.207,-178.136,6.872,148.727
C02555=1166.735,182.378,-59.184,-178.140,6.869,148.727
C02556=1166.739,182.129,-59.161,-178.142,6.867,148.728
C02557=1166.744,181.880,-59.138,-178.144,6.865,148.728
C02558=1166.749,181.630,-59.115,-178.147,6.863,148.728
C02559=1166.753,181.382,-59.092,-178.150,6.861,148.729
C02560=1166.758,181.133,-59.069,-178.153,6.859,148.729
C02561=1166.762,180.885,-59.046,-178.156,6.857,148.729
C02562=1166.767,180.635,-59.024,-178.158,6.855,148.730
C02563=1166.772,180.386,-59.000,-178.161,6.853,148.730
C02564=1166.776,180.138,-58.978,-178.164,6.851,148.730
C02565=1166.781,179.888,-58.955,-178.167,6.849,148.731
C02566=1166.785,179.640,-58.933,-178.169,6.847,148.731
C02567=1166.790,179.391,-58.909,-178.172,6.845,148.731
C02568=1166.795,179.142,-58.888,-178.175,6.843,148.731
C02569=1166.799,178.893,-58.864,-178.177,6.841,148.732
C02570=1166.803,178.644,-58.842,-178.180,6.839,148.732
C02571=1166.808,178.394,-58.819,-178.183,6.837,148.733
C02572=1166.813,178.146,-58.796,-178.186,6.834,148.733
C02573=1166.818,177.897,-58.774,-178.188,6.833,148.733
C02574=1166.822,177.648,-58.751,-178.191,6.831,148.733
C02575=1166.827,177.400,-58.728,-178.194,6.829,148.734
C02576=1166.832,177.150,-58.706,-178.196,6.827,148.734
C02577=1166.836,176.901,-58.683,-178.199,6.825,148.734
C02578=1166.841,176.652,-58.661,-178.202,6.823,148.735
C02579=1166.846,176.404,-58.638,-178.204,6.821,148.735
C02580=1166.850,176.154,-58.616,-178.207,6.819,148.735
C02581=1166.855,175.905,-58.592,-178.210,6.817,148.736
C02582=1166.860,175.657,-58.571,-178.213,6.815,148.736
C02583=1166.864,175.408,-58.547,-178.215,6.813,148.736
C02584=1166.869,175.158,-58.525,-178.218,6.811,148.737
C02585=1166.873,174.910,-58.503,-178.221,6.809,148.737
C02586=1166.878,174.661,-58.480,-178.223,6.808,148.737
C02587=1166.883,174.412,-58.458,-178.227,6.805,148.738
C02588=1166.888,174.163,-58.435,-178.229,6.803,148.738
C02589=1166.892,173.914,-58.413,-178.232,6.801,148.738
C02590=1166.897,173.666,-58.391,-178.234,6.799,148.738
C02591=1166.902,173.416,-58.368,-178.237,6.798,148.739
C02592=1166.906,173.167,-58.346,-178.240,6.796,148.739
C02593=1166.910,172.919,-58.324,-178.243,6.793,148.740
C02594=1166.915,172.669,-58.301,-178.246,6.791,148.740
C02595=1166.920,172.420,-58.279,-178.248,6.790,148.740
C02596=1166.924,172.172,-58.256,-178.250,6.788,148.740
C02597=1166.929,171.922,-58.234,-178.253,6.786,148.741
C02598=1166.934,171.673,-58.212,-178.256,6.783,148.741
C02599=1166.938,171.425,-58.189,-178.259,6.782,148.741
C02600=1166.944,171.176,-58.167,-178.262,6.780,148.742
C02601=1166.948,170.926,-58.145,-178.264,6.778,148.742
C02602=1166.953,170.678,-58.123,-178.267,6.776,148.743
C02603=1166.958,170.429,-58.100,-178.269,6.774,148.743
C02604=1166.962,170.179,-58.078,-178.273,6.772,148.743
C02605=1166.967,169.931,-58.056,-178.275,6.770,148.743
C02606=1166.971,169.681,-58.034,-178.278,6.768,148.744
C02607=1166.976,169.433,-58.011,-178.281,6.766,148.744
C02608=1166.981,169.184,-57.989,-178.283,6.765,148.745
C02609=1166.985,168.935,-57.967,-178.286,6.763,148.745
C02610=1166.990,168.686,-57.945,-178.289,6.761,148.745
C02611=1166.995,168.437,-57.923,-178.292,6.758,148.745
C02612=1167.000,168.187,-57.901,-178.294,6.756,148.746
C02613=1167.004,167.939,-57.879,-178.297,6.755,148.746
C02614=1167.008,167.690,-57.857,-178.300,6.753,148.747
C02615=1167.013,167.441,-57.835,-178.302,6.751,148.747
C02616=1167.018,167.192,-57.813,-178.305,6.749,148.747
C02617=1167.023,166.943,-57.791,-178.308,6.748,148.748
C02618=1167.027,166.694,-57.769,-178.311,6.745,148.748
C02619=1167.032,166.445,-57.747,-178.314,6.743,148.748
C02620=1167.037,166.196,-57.725,-178.316,6.741,148.749
C02621=1167.041,165.947,-57.703,-178.319,6.739,148.749
C02622=1167.046,165.698,-57.681,-178.321,6.738,148.749
C02623=1167.051,165.449,-57.659,-178.324,6.736,148.750
C02624=1167.056,165.199,-57.637,-178.327,6.734,148.750
C02625=1167.060,164.951,-57.615,-178.329,6.732,148.750
C02626=1167.065,164.701,-57.593,-178.333,6.730,148.751
C02627=1167.070,164.453,-57.571,-178.335,6.728,148.751
C02628=1167.074,164.204,-57.550,-178.338,6.726,148.751
C02629=1167.079,163.955,-57.528,-178.341,6.725,148.752
C02630=1167.084,163.706,-57.506,-178.343,6.723,148.752
C02631=1167.088,163.457,-57.484,-178.346,6.721,148.752
C02632=1167.093,163.208,-57.462,-178.348,6.719,148.753
C02633=1167.097,162.959,-57.440,-178.351,6.717,148.753
C02634=1167.102,162.710,-57.419,-178.354,6.715,148.753
C02635=1167.107,162.462,-57.397,-178.357,6.713,148.754
C02636=1167.111,162.212,-57.375,-178.360,6.711,148.754
C02637=1167.116,161.963,-57.354,-178.362,6.709,148.755
C02638=1167.120,161.714,-57.332,-178.365,6.708,148.755
C02639=1167.125,161.465,-57.310,-178.368,6.706,148.755
C02640=1167.130,161.216,-57.288,-178.370,6.704,148.756
C02641=1167.134,160.967,-57.266,-178.373,6.702,148.756
C02642=1167.140,160.718,-57.245,-178.376,6.701,148.756
C02643=1167.144,160.469,-57.224,-178.378,6.699,148.757
C02644=1167.149,160.220,-57.202,-178.381,6.697,148.757
C02645=1167.154,159.971,-57.180,-178.383,6.695,148.757
C02646=1167.158,159.722,-57.158,-178.387,6.692,148.758
C02647=1167.163,159.473,-57.137,-178.389,6.691,148.758
C02648=1167.168,159.224,-57.115,-178.392,6.689,148.758
C02649=1167.172,158.975,-57.093,-178.395,6.687,148.759
C02650=1167.177,158.725,-57.072,-178.397,6.685,148.759
C02651=1167.182,158.457,-57.049,-178.400,6.684,148.760
C02652=1167.187,158.188,-57.025,-178.403,6.681,148.760
C02653=1167.192,157.918,-57.003,-178.407,6.680,148.761
C02654=1167.197,157.650,-56.979,-178.409,6.678,148.761
C02655=1167.202,157.400,-56.958,-178.412,6.676,148.761
C02656=1167.206,157.152,-56.937,-178.415,6.675,148.762
C02657=1167.212,156.903,-56.916,-178.417,6.673,148.762
C02658=1167.216,156.654,-56.894,-178.420,6.671,148.762
C02659=1167.221,156.405,-56.872,-178.423,6.669,148.763
C02660=1167.226,156.156,-56.851,-178.426,6.667,148.763
C02661=1167.230,155.906,-56.829,-178.428,6.665,148.763
C02662=1167.235,155.657,-56.808,-178.431,6.663,148.764
C02663=1167.240,155.409,-56.787,-178.434,6.661,148.764
C02664=1167.244,155.160,-56.765,-178.436,6.659,148.764
C02665=1167.249,154.910,-56.744,-178.439,6.658,148.765
C02666=1167.254,154.661,-56.722,-178.442,6.656,148.765
C02667=1167.259,154.412,-56.701,-178.444,6.654,148.766
C02668=1167.263,154.164,-56.680,-178.447,6.652,148.766
C02669=1167.268,153.914,-56.659,-178.450,6.651,148.766
C02670=1167.273,153.665,-56.637,-178.452,6.649,148.767
C02671=1167.278,153.416,-56.616,-178.455,6.647,148.767
C02672=1167.282,153.168,-56.595,-178.458,6.645,148.767
C02673=1167.286,152.918,-56.574,-178.461,6.644,148.768
C02674=1167.292,152.668,-56.553,-178.463,6.642,148.768
C02675=1167.297,152.420,-56.531,-178.466,6.640,148.769
C02676=1167.301,152.171,-56.511,-178.469,6.638,148.769
C02677=1167.306,151.922,-56.489,-178.471,6.637,148.769
C02678=1167.310,151.672,-56.468,-178.474,6.635,148.770
C02679=1167.315,151.423,-56.447,-178.477,6.633,148.770
C02680=1167.320,151.175,-56.426,-178.479,6.631,148.770
C02681=1167.325,150.925,-56.405,-178.482,6.630,148.771
C02682=1167.329,150.677,-56.383,-178.485,6.628,148.771
C02683=1167.334,150.428,-56.362,-178.487,6.626,148.772
C02684=1167.339,150.178,-56.341,-178.490,6.624,148.772
C02685=1167.343,149.929,-56.321,-178.493,6.623,148.772
C02686=1167.348,149.680,-56.299,-178.496,6.621,148.773
C02687=1167.353,149.431,-56.278,-178.498,6.619,148.773
C02688=1167.358,149.182,-56.258,-178.501,6.617,148.774
C02689=1167.363,148.933,-56.236,-178.504,6.616,148.774
C02690=1167.367,148.683,-56.215,-178.506,6.614,148.774
C02691=1167.372,148.435,-56.194,-178.510,6.613,148.775
C02692=1167.377,148.185,-56.173,-178.512,6.611,148.775
C02693=1167.381,147.937,-56.152,-178.515,6.609,148.776
C02694=1167.386,147.688,-56.131,-178.518,6.607,148.776
C02695=1167.390,147.439,-56.111,-178.520,6.606,148.776
C02696=1167.396,147.189,-56.090,-178.523,6.604,148.777
C02697=1167.401,146.940,-56.069,-178.526,6.602,148.777
C02698=1167.405,146.692,-56.048,-178.528,6.600,148.778
C02699=1167.410,146.442,-56.027,-178.531,6.599,148.778
C02700=1167.414,146.193,-56.006,-178.534,6.597,148.778
C02701=1167.419,145.944,-55.985,-178.537,6.595,148.779
C02702=1167.424,145.695,-55.965,-178.539,6.593,148.779
C02703=1167.429,145.446,-55.944,-178.542,6.592,148.779
C02704=1167.433,145.197,-55.924,-178.545,6.590,148.780
C02705=1167.438,144.947,-55.903,-178.547,6.588,148.780
C02706=1167.443,144.699,-55.882,-178.550,6.586,148.781
C02707=1167.448,144.450,-55.861,-178.553,6.585,148.781
C02708=1167.452,144.201,-55.840,-178.555,6.583,148.781
C02709=1167.457,143.952,-55.819,-178.558,6.581,148.782
C02710=1167.462,143.703,-55.799,-178.561,6.580,148.782
C02711=1167.467,143.453,-55.778,-178.563,6.578,148.783
C02712=1167.471,143.204,-55.758,-178.566,6.576,148.783
C02713=1167.476,142.955,-55.737,-178.569,6.575,148.784
C02714=1167.481,142.706,-55.716,-178.572,6.573,148.784
C02715=1167.485,142.457,-55.696,-178.575,6.571,148.784
C02716=1167.490,142.207,-55.674,-178.577,6.569,148.785
C02717=1167.494,141.958,-55.654,-178.580,6.568,148.785
C02718=1167.500,141.709,-55.633,-178.583,6.566,148.785
C02719=1167.504,141.460,-55.613,-178.586,6.564,148.786
C02720=1167.508,141.211,-55.592,-178.588,6.562,148.786
C02721=1167.514,140.962,-55.571,-178.591,6.561,148.787
C02722=1167.518,140.712,-55.552,-178.594,6.559,148.787
C02723=1167.523,140.463,-55.531,-178.596,6.557,148.787
C02724=1167.529,140.215,-55.511,-178.599,6.556,148.788
C02725=1167.533,139.966,-55.490,-178.601,6.555,148.788
C02726=1167.537,139.717,-55.470,-178.604,6.553,148.789
C02727=1167.543,139.468,-55.449,-178.607,6.552,148.789
C02728=1167.547,139.219,-55.429,-178.610,6.550,148.790
C02729=1167.552,138.970,-55.408,-178.612,6.548,148.790
C02730=1167.557,138.720,-55.388,-178.615,6.546,148.790
C02731=1167.561,138.471,-55.368,-178.618,6.545,148.791
C02732=1167.566,138.222,-55.347,-178.621,6.543,148.791
C02733=1167.571,137.973,-55.326,-178.623,6.541,148.792
C02734=1167.575,137.724,-55.306,-178.626,6.539,148.792
C02735=1167.580,137.474,-55.286,-178.629,6.538,148.792
C02736=1167.585,137.225,-55.266,-178.631,6.536,148.793
C02737=1167.590,136.976,-55.245,-178.635,6.534,148.793
C02738=1167.594,136.727,-55.225,-178.637,6.533,148.794
C02739=1167.599,136.477,-55.205,-178.639,6.532,148.794
C02740=1167.604,136.229,-55.185,-178.642,6.530,148.794
C02741=1167.609,135.980,-55.164,-178.645,6.528,148.795
C02742=1167.614,135.730,-55.144,-178.648,6.527,148.795
C02743=1167.618,135.481,-55.124,-178.650,6.525,148.796
C02744=1167.623,135.232,-55.104,-178.653,6.523,148.796
C02745=1167.628,134.983,-55.084,-178.656,6.521,148.796
C02746=1167.633,134.734,-55.063,-178.659,6.520,148.797
C02747=1167.637,134.485,-55.043,-178.662,6.518,148.797
C02748=1167.642,134.235,-55.023,-178.664,6.517,148.798
C02749=1167.647,133.987,-55.003,-178.667,6.515,148.798
C02750=1167.652,133.737,-54.983,-178.669,6.514,148.799
C02751=1167.657,133.488,-54.962,-178.672,6.512,148.799
C02752=1167.661,133.239,-54.942,-178.674,6.510,148.799
C02753=1167.666,132.990,-54.922,-178.677,6.509,148.800
C02754=1167.671,132.741,-54.902,-178.680,6.507,148.800
C02755=1167.675,132.472,-54.881,-178.683,6.506,148.801
C02756=1167.681,132.203,-54.859,-178.686,6.504,148.801
C02757=1167.686,131.935,-54.837,-178.688,6.502,148.802
C02758=1167.691,131.666,-54.816,-178.692,6.501,148.802
C02759=1167.696,131.418,-54.796,-178.694,6.499,148.803
C02760=1167.701,131.168,-54.776,-178.697,6.497,148.803
C02761=1167.706,130.919,-54.756,-178.700,6.496,148.803
C02762=1167.710,130.670,-54.736,-178.702,6.494,148.804
C02763=1167.715,130.421,-54.716,-178.705,6.492,148.804
C02764=1167.720,130.172,-54.696,-178.708,6.491,148.805
C02765=1167.725,129.922,-54.677,-178.711,6.489,148.805
C02766=1167.729,129.673,-54.656,-178.713,6.488,148.806
C02767=1167.734,129.424,-54.637,-178.716,6.486,148.806
C02768=1167.740,129.175,-54.616,-178.719,6.485,148.806
C02769=1167.745,128.926,-54.596,-178.721,6.483,148.807
C02770=1167.749,128.676,-54.577,-178.724,6.481,148.807
C02771=1167.754,128.427,-54.556,-178.727,6.480,148.808
C02772=1167.759,128.178,-54.537,-178.730,6.478,148.808
C02773=1167.763,127.929,-54.517,-178.732,6.477,148.809
C02774=1167.768,127.680,-54.497,-178.735,6.475,148.809
C02775=1167.773,127.430,-54.477,-178.737,6.474,148.809
C02776=1167.777,127.182,-54.458,-178.740,6.472,148.810
C02777=1167.782,126.933,-54.438,-178.743,6.471,148.810
C02778=1167.787,126.683,-54.419,-178.746,6.469,148.811
C02779=1167.792,126.434,-54.399,-178.749,6.467,148.811
C02780=1167.797,126.185,-54.379,-178.751,6.466,148.812
C02781=1167.801,125.936,-54.359,-178.754,6.465,148.812
C02782=1167.806,125.686,-54.340,-178.756,6.463,148.812
C02783=1167.811,125.438,-54.320,-178.760,6.461,148.813
C02784=1167.816,125.188,-54.300,-178.762,6.460,148.813
C02785=1167.821,124.939,-54.280,-178.765,6.458,148.814
C02786=1167.825,124.689,-54.261,-178.767,6.457,148.814
C02787=1167.831,124.440,-54.241,-178.770,6.455,148.815
C02788=1167.835,124.191,-54.221,-178.773,6.454,148.815
C02789=1167.839,123.942,-54.202,-178.776,6.452,148.816
C02790=1167.844,123.693,-54.183,-178.778,6.450,148.816
C02791=1167.849,123.444,-54.163,-178.781,6.449,148.816
C02792=1167.854,123.194,-54.143,-178.783,6.448,148.817
C02793=1167.859,122.945,-54.124,-178.786,6.446,148.817
C02794=1167.864,122.696,-54.104,-178.789,6.445,148.818
C02795=1167.868,122.447,-54.085,-178.792,6.443,148.818
C02796=1167.873,122.198,-54.065,-178.795,6.441,148.819
C02797=1167.878,121.949,-54.046,-178.797,6.440,148.819
C02798=1167.883,121.700,-54.026,-178.799,6.439,148.819
C02799=1167.888,121.450,-54.007,-178.803,6.437,148.820
C02800=1167.893,121.201,-53.987,-178.805,6.436,148.820
C02801=1167.897,120.952,-53.968,-178.808,6.434,148.821
C02802=1167.902,120.702,-53.949,-178.811,6.432,148.821
C02803=1167.907,120.454,-53.929,-178.813,6.431,148.822
C02804=1167.912,120.204,-53.910,-178.816,6.430,148.822
C02805=1167.916,119.955,-53.891,-178.819,6.428,148.823
C02806=1167.921,119.706,-53.871,-178.821,6.426,148.823
C02807=1167.926,119.456,-53.852,-178.824,6.425,148.823
C02808=1167.931,119.207,-53.833,-178.827,6.424,148.824
C02809=1167.935,118.958,-53.813,-178.829,6.422,148.825
C02810=1167.940,118.709,-53.794,-178.832,6.421,148.825
C02811=1167.946,118.460,-53.774,-178.835,6.419,148.825
C02812=1167.950,118.210,-53.755,-178.838,6.417,148.826
C02813=1167.955,117.962,-53.736,-178.840,6.417,148.826
C02814=1167.960,117.712,-53.716,-178.843,6.415,148.827
C02815=1167.965,117.463,-53.697,-178.846,6.413,148.827
C02816=1167.969,117.214,-53.678,-178.848,6.412,148.828
C02817=1167.974,116.965,-53.659,-178.851,6.411,148.828
C02818=1167.979,116.716,-53.639,-178.854,6.409,148.829
C02819=1167.983,116.466,-53.621,-178.856,6.408,148.829
C02820=1167.989,116.217,-53.602,-178.859,6.406,148.829
C02821=1167.994,115.967,-53.582,-178.862,6.404,148.830
C02822=1167.998,115.719,-53.563,-178.864,6.404,148.830
C02823=1168.003,115.469,-53.544,-178.867,6.402,148.831
C02824=1168.008,115.220,-53.524,-178.870,6.400,148.831
C02825=1168.013,114.970,-53.506,-178.873,6.398,148.832
C02826=1168.018,114.721,-53.487,-178.875,6.398,148.832
C02827=1168.022,114.472,-53.468,-178.878,6.396,148.833
C02828=1168.027,114.223,-53.448,-178.881,6.394,148.833
C02829=1168.032,113.974,-53.429,-178.883,6.393,148.833
C02830=1168.037,113.725,-53.411,-178.886,6.392,148.834
C02831=1168.042,113.476,-53.391,-178.889,6.390,148.835
C02832=1168.046,113.226,-53.372,-178.891,6.389,148.835
C02833=1168.052,112.977,-53.354,-178.894,6.387,148.835
C02834=1168.057,112.727,-53.334,-178.897,6.386,148.836
C02835=1168.061,112.479,-53.315,-178.899,6.385,148.836
C02836=1168.066,112.229,-53.296,-178.902,6.383,148.837
C02837=1168.071,111.980,-53.278,-178.905,6.381,148.837
C02838=1168.076,111.731,-53.258,-178.907,6.381,148.838
C02839=1168.080,111.482,-53.239,-178.910,6.379,148.838
C02840=1168.085,111.232,-53.220,-178.913,6.377,148.839
C02841=1168.090,110.983,-53.202,-178.916,6.376,148.839
C02842=1168.096,110.734,-53.183,-178.918,6.375,148.840
C02843=1168.100,110.485,-53.164,-178.921,6.373,148.840
C02844=1168.105,110.236,-53.145,-178.924,6.372,148.841
C02845=1168.109,109.986,-53.126,-178.926,6.370,148.841
C02846=1168.115,109.737,-53.107,-178.929,6.369,148.842
C02847=1168.119,109.488,-53.089,-178.932,6.368,148.842
C02848=1168.124,109.238,-53.070,-178.934,6.366,148.842
C02849=1168.129,108.990,-53.051,-178.937,6.365,148.843
C02850=1168.133,108.740,-53.032,-178.940,6.364,148.843
C02851=1168.138,108.491,-53.013,-178.942,6.362,148.844
C02852=1168.143,108.242,-52.995,-178.945,6.360,148.844
C02853=1168.148,107.992,-52.976,-178.948,6.360,148.845
C02854=1168.153,107.743,-52.958,-178.950,6.358,148.845
C02855=1168.158,107.493,-52.938,-178.953,6.356,148.846
C02856=1168.163,107.244,-52.920,-178.955,6.355,148.846
C02857=1168.167,106.996,-52.901,-178.959,6.354,148.847
C02858=1168.172,106.745,-52.882,-178.961,6.352,148.847
C02859=1168.177,106.478,-52.862,-178.964,6.351,148.848
C02860=1168.183,106.209,-52.842,-178.967,6.349,148.848
C02861=1168.188,105.941,-52.823,-178.970,6.347,148.849
C02862=1168.193,105.672,-52.802,-178.973,6.346,148.849
C02863=1168.198,105.423,-52.784,-178.975,6.345,148.850
C02864=1168.203,105.174,-52.765,-178.978,6.343,148.850
C02865=1168.207,104.924,-52.746,-178.981,6.342,148.851
C02866=1168.212,104.675,-52.728,-178.983,6.341,148.851
C02867=1168.217,104.426,-52.710,-178.986,6.339,148.852
C02868=1168.222,104.177,-52.690,-178.989,6.338,148.852
C02869=1168.227,103.927,-52.672,-178.991,6.337,148.853
C02870=1168.232,103.678,-52.654,-178.994,6.336,148.853
C02871=1168.237,103.429,-52.635,-178.997,6.334,148.853
C02872=1168.242,103.179,-52.617,-178.999,6.333,148.854
C02873=1168.246,102.930,-52.599,-179.002,6.332,148.854
C02874=1168.252,102.681,-52.580,-179.005,6.330,148.855
C02875=1168.256,102.431,-52.561,-179.008,6.328,148.855
C02876=1168.261,102.182,-52.543,-179.010,6.328,148.856
C02877=1168.266,101.934,-52.525,-179.013,6.326,148.856
C02878=1168.271,101.684,-52.506,-179.016,6.325,148.857
C02879=1168.276,101.434,-52.488,-179.018,6.324,148.857
C02880=1168.280,101.185,-52.470,-179.021,6.322,148.858
C02881=1168.285,100.937,-52.451,-179.024,6.321,148.858
C02882=1168.290,100.688,-52.433,-179.026,6.320,148.859
C02883=1168.295,100.437,-52.414,-179.029,6.318,148.859
C02884=1168.300,100.188,-52.396,-179.032,6.316,148.860
C02885=1168.305,99.939,-52.378,-179.034,6.316,148.860
C02886=1168.310,99.690,-52.360,-179.037,6.314,148.861
C02887=1168.314,99.441,-52.341,-179.040,6.312,148.861
C02888=1168.319,99.191,-52.322,-179.042,6.312,148.862
C02889=1168.324,98.942,-52.304,-179.045,6.310,148.862
C02890=1168.329,98.693,-52.287,-179.047,6.309,148.863
C02891=1168.334,98.444,-52.269,-179.050,6.308,148.863
C02892=1168.338,98.194,-52.250,-179.053,6.306,148.864
C02893=1168.343,97.944,-52.232,-179.055,6.305,148.864
C02894=1168.348,97.696,-52.214,-179.058,6.304,148.865
C02895=1168.354,97.446,-52.195,-179.061,6.302,148.865
C02896=1168.359,97.197,-52.177,-179.063,6.301,148.866
C02897=1168.363,96.948,-52.159,-179.067,6.300,148.866
C02898=1168.368,96.698,-52.141,-179.069,6.298,148.867
C02899=1168.373,96.449,-52.123,-179.071,6.297,148.867
C02900=1168.378,96.200,-52.105,-179.075,6.296,148.868
C02901=1168.383,95.951,-52.087,-179.077,6.294,148.868
C02902=1168.387,95.701,-52.069,-179.079,6.293,148.868
C02903=1168.392,95.452,-52.051,-179.083,6.292,148.869
C02904=1168.397,95.203,-52.033,-179.085,6.291,148.870
C02905=1168.402,94.953,-52.014,-179.088,6.289,148.870
C02906=1168.406,94.704,-51.996,-179.091,6.288,148.871
C02907=1168.412,94.455,-51.978,-179.093,6.287,148.871
C02908=1168.417,94.205,-51.960,-179.096,6.285,148.871
C02909=1168.422,93.956,-51.942,-179.099,6.284,148.872
C02910=1168.427,93.707,-51.924,-179.101,6.283,148.873
C02911=1168.432,93.458,-51.906,-179.104,6.282,148.873
C02912=1168.437,93.208,-51.889,-179.106,6.281,148.874
C02913=1168.441,92.958,-51.870,-179.109,6.279,148.874
C02914=1168.446,92.709,-51.852,-179.112,6.278,148.875
C02915=1168.451,92.460,-51.834,-179.114,6.277,148.875
C02916=1168.456,92.211,-51.816,-179.117,6.275,148.875
C02917=1168.461,91.962,-51.798,-179.120,6.275,148.876
C02918=1168.465,91.713,-51.781,-179.122,6.273,148.877
C02919=1168.470,91.463,-51.763,-179.125,6.271,148.877
C02920=1168.475,91.214,-51.746,-179.128,6.271,148.878
C02921=1168.480,90.965,-51.728,-179.131,6.269,148.878
C02922=1168.485,90.715,-51.710,-179.133,6.267,148.878
C02923=1168.490,90.466,-51.692,-179.136,6.267,148.879
C02924=1168.495,90.217,-51.674,-179.139,6.265,148.880
C02925=1168.500,89.967,-51.657,-179.141,6.265,148.880
C02926=1168.504,89.717,-51.638,-179.144,6.263,148.881
C02927=1168.509,89.468,-51.620,-179.146,6.262,148.881
C02928=1168.514,89.219,-51.602,-179.149,6.261,148.882
C02929=1168.519,88.969,-51.585,-179.152,6.259,148.882
C02930=1168.524,88.720,-51.567,-179.154,6.258,148.882
C02931=1168.529,88.471,-51.550,-179.157,6.257,148.883
C02932=1168.533,88.222,-51.532,-179.159,6.256,148.884
C02933=1168.539,87.972,-51.514,-179.162,6.254,148.884
C02934=1168.544,87.723,-51.496,-179.165,6.253,148.885
C02935=1168.549,87.474,-51.478,-179.168,6.252,148.885
C02936=1168.554,87.224,-51.461,-179.171,6.251,148.886
C02937=1168.559,86.975,-51.443,-179.173,6.250,148.886
C02938=1168.563,86.726,-51.426,-179.176,6.248,148.887
C02939=1168.568,86.476,-51.409,-179.178,6.248,148.887
C02940=1168.573,86.227,-51.391,-179.181,6.246,148.888
C02941=1168.578,85.978,-51.373,-179.184,6.244,148.888
C02942=1168.583,85.728,-51.355,-179.186,6.244,148.889
C02943=1168.587,85.479,-51.338,-179.189,6.242,148.889
C02944=1168.592,85.229,-51.321,-179.192,6.241,148.890
C02945=1168.598,84.981,-51.303,-179.194,6.240,148.890
C02946=1168.603,84.732,-51.285,-179.197,6.239,148.891
C02947=1168.607,84.482,-51.268,-179.200,6.237,148.891
C02948=1168.612,84.233,-51.250,-179.203,6.236,148.892
C02949=1168.618,83.983,-51.233,-179.205,6.235,148.892
C02950=1168.622,83.734,-51.215,-179.208,6.234,148.893
C02951=1168.627,83.485,-51.199,-179.210,6.233,148.893
C02952=1168.632,83.235,-51.181,-179.213,6.231,148.894
C02953=1168.637,82.986,-51.163,-179.215,6.230,148.894
C02954=1168.642,82.736,-51.145,-179.219,6.229,148.895
C02955=1168.646,82.487,-51.129,-179.221,6.228,148.895
C02956=1168.651,82.238,-51.111,-179.223,6.226,148.896
C02957=1168.657,81.988,-51.093,-179.226,6.226,148.896
C02958=1168.661,81.739,-51.076,-179.229,6.224,148.897
C02959=1168.667,81.490,-51.059,-179.232,6.223,148.897
C02960=1168.671,81.241,-51.041,-179.234,6.222,148.898
C02961=1168.676,80.991,-51.024,-179.237,6.220,148.898
C02962=1168.681,80.742,-51.007,-179.239,6.220,148.899
C02963=1168.686,80.473,-50.988,-179.242,6.218,148.899
C02964=1168.692,80.205,-50.969,-179.245,6.217,148.900
C02965=1168.697,79.937,-50.951,-179.248,6.216,148.901
C02966=1168.702,79.668,-50.933,-179.251,6.215,148.901
C02967=1168.707,79.419,-50.915,-179.254,6.213,148.902
C02968=1168.712,79.169,-50.898,-179.256,6.212,148.902
C02969=1168.717,78.921,-50.880,-179.259,6.211,148.903
C02970=1168.722,78.671,-50.864,-179.262,6.210,148.903
C02971=1168.727,78.421,-50.846,-179.264,6.208,148.904
C02972=1168.732,78.172,-50.829,-179.267,6.208,148.904
C02973=1168.736,77.923,-50.812,-179.270,6.206,148.905
C02974=1168.741,77.673,-50.795,-179.272,6.206,148.905
C02975=1168.747,77.424,-50.778,-179.275,6.204,148.906
C02976=1168.751,77.175,-50.760,-179.277,6.203,148.906
C02977=1168.757,76.925,-50.743,-179.280,6.202,148.907
C02978=1168.761,76.676,-50.726,-179.282,6.201,148.907
C02979=1168.766,76.426,-50.709,-179.286,6.200,148.908
C02980=1168.771,76.178,-50.692,-179.288,6.199,148.908
C02981=1168.776,75.928,-50.675,-179.291,6.197,148.909
C02982=1168.781,75.678,-50.658,-179.293,6.197,148.910
C02983=1168.786,75.429,-50.641,-179.296,6.195,148.910
C02984=1168.790,75.180,-50.623,-179.299,6.194,148.911
C02985=1168.796,74.931,-50.607,-179.301,6.193,148.911
C02986=1168.801,74.681,-50.590,-179.304,6.192,148.912
C02987=1168.806,74.431,-50.573,-179.307,6.190,148.912
C02988=1168.810,74.182,-50.556,-179.309,6.190,148.913
C02989=1168.815,73.932,-50.539,-179.312,6.188,148.913
C02990=1168.821,73.683,-50.522,-179.315,6.188,148.914
C02991=1168.825,73.434,-50.504,-179.317,6.186,148.914
C02992=1168.830,73.185,-50.488,-179.319,6.185,148.915
C02993=1168.835,72.935,-50.470,-179.323,6.184,148.915
C02994=1168.840,72.686,-50.454,-179.325,6.183,148.916
C02995=1168.845,72.437,-50.438,-179.328,6.182,148.916
C02996=1168.850,72.187,-50.420,-179.330,6.181,148.917
C02997=1168.855,71.938,-50.404,-179.333,6.180,148.918
C02998=1168.860,71.688,-50.387,-179.336,6.178,148.918
C02999=1168.865,71.439,-50.370,-179.338,6.178,148.918
C03000=1168.870,71.189,-50.353,-179.341,6.176,148.919
C03001=1168.875,70.940,-50.336,-179.343,6.175,148.920
C03002=1168.880,70.691,-50.320,-179.346,6.174,148.920
C03003=1168.885,70.441,-50.303,-179.348,6.173,148.921
C03004=1168.890,70.192,-50.286,-179.352,6.172,148.921
C03005=1168.894,69.943,-50.270,-179.354,6.171,148.922
C03006=1168.899,69.693,-50.252,-179.357,6.170,148.922
C03007=1168.904,69.443,-50.236,-179.359,6.169,148.923
C03008=1168.910,69.194,-50.219,-179.362,6.167,148.923
C03009=1168.914,68.945,-50.202,-179.365,6.167,148.924
C03010=1168.919,68.695,-50.185,-179.367,6.165,148.924
C03011=1168.925,68.446,-50.168,-179.370,6.164,148.925
C03012=1168.929,68.197,-50.152,-179.372,6.163,148.925
C03013=1168.934,67.947,-50.135,-179.375,6.162,148.926
C03014=1168.939,67.698,-50.119,-179.377,6.161,148.927
C03015=1168.944,67.449,-50.102,-179.381,6.160,148.927
C03016=1168.948,67.199,-50.085,-179.383,6.159,148.928
C03017=1168.953,66.950,-50.069,-179.386,6.158,148.928
C03018=1168.959,66.701,-50.051,-179.388,6.157,148.929
C03019=1168.964,66.451,-50.036,-179.391,6.156,148.929
C03020=1168.968,66.202,-50.019,-179.394,6.155,148.930
C03021=1168.973,65.952,-50.002,-179.396,6.154,148.930
C03022=1168.979,65.703,-49.986,-179.399,6.152,148.931
C03023=1168.983,65.454,-49.969,-179.402,6.152,148.932
C03024=1168.988,65.204,-49.952,-179.404,6.150,148.932
C03025=1168.993,64.955,-49.937,-179.406,6.149,148.932
C03026=1168.998,64.705,-49.919,-179.410,6.148,148.933
C03027=1169.003,64.456,-49.903,-179.412,6.147,148.934
C03028=1169.008,64.207,-49.886,-179.414,6.147,148.934
C03029=1169.012,63.957,-49.870,-179.417,6.145,148.935
C03030=1169.019,63.707,-49.853,-179.420,6.145,148.935
C03031=1169.023,63.458,-49.837,-179.423,6.143,148.936
C03032=1169.028,63.209,-49.821,-179.425,6.142,148.936
C03033=1169.033,62.959,-49.805,-179.428,6.141,148.937
C03034=1169.038,62.710,-49.788,-179.431,6.140,148.937
C03035=1169.042,62.461,-49.772,-179.433,6.139,148.938
C03036=1169.048,62.211,-49.754,-179.436,6.138,148.939
C03037=1169.053,61.962,-49.739,-179.438,6.137,148.939
C03038=1169.058,61.712,-49.722,-179.441,6.136,148.940
C03039=1169.063,61.463,-49.706,-179.443,6.135,148.940
C03040=1169.067,61.213,-49.690,-179.446,6.134,148.941
C03041=1169.072,60.964,-49.674,-179.449,6.133,148.941
C03042=1169.077,60.715,-49.657,-179.451,6.132,148.942
C03043=1169.083,60.465,-49.641,-179.454,6.131,148.942
C03044=1169.088,60.216,-49.624,-179.457,6.130,148.943
C03045=1169.093,59.967,-49.608,-179.459,6.129,148.943
C03046=1169.097,59.717,-49.592,-179.462,6.128,148.944
C03047=1169.102,59.468,-49.575,-179.464,6.127,148.944
C03048=1169.107,59.218,-49.559,-179.468,6.126,148.945
C03049=1169.112,58.969,-49.543,-179.470,6.125,148.946
C03050=1169.117,58.719,-49.527,-179.472,6.124,148.946
C03051=1169.122,58.470,-49.511,-179.475,6.123,148.947
C03052=1169.127,58.221,-49.494,-179.478,6.122,148.947
C03053=1169.132,57.971,-49.479,-179.480,6.120,148.948
C03054=1169.137,57.722,-49.462,-179.483,6.120,148.948
C03055=1169.143,57.472,-49.446,-179.485,6.119,148.949
C03056=1169.147,57.223,-49.429,-179.488,6.118,148.950
C03057=1169.153,56.973,-49.414,-179.491,6.117,148.950
C03058=1169.157,56.724,-49.397,-179.493,6.116,148.951
C03059=1169.162,56.474,-49.381,-179.496,6.115,148.951
C03060=1169.167,56.225,-49.365,-179.499,6.114,148.952
C03061=1169.172,55.976,-49.349,-179.501,6.112,148.952
C03062=1169.177,55.726,-49.332,-179.504,6.112,148.953
C03063=1169.182,55.477,-49.317,-179.506,6.111,148.953
C03064=1169.188,55.227,-49.301,-179.509,6.110,148.954
C03065=1169.192,54.978,-49.285,-179.512,6.109,148.954
C03066=1169.197,54.728,-49.269,-179.514,6.108,148.955
C03067=1169.202,54.459,-49.252,-179.517,6.107,148.956
C03068=1169.208,54.191,-49.234,-179.520,6.106,148.956
C03069=1169.213,53.923,-49.217,-179.523,6.105,148.957
C03070=1169.219,53.654,-49.200,-179.526,6.103,148.957
C03071=1169.224,53.404,-49.184,-179.528,6.103,148.958
C03072=1169.229,53.156,-49.168,-179.530,6.102,148.958
C03073=1169.233,52.906,-49.152,-179.534,6.101,148.959
C03074=1169.238,52.656,-49.137,-179.536,6.100,148.959
C03075=1169.243,52.408,-49.120,-179.538,6.099,148.960
C03076=1169.248,52.157,-49.104,-179.541,6.098,148.961
C03077=1169.253,51.908,-49.089,-179.544,6.097,148.961
C03078=1169.258,51.659,-49.072,-179.546,6.096,148.962
C03079=1169.263,51.409,-49.056,-179.549,6.095,148.962
C03080=1169.269,51.160,-49.041,-179.552,6.094,148.963
C03081=1169.273,50.910,-49.025,-179.554,6.093,148.963
C03082=1169.278,50.661,-49.009,-179.557,6.092,148.964
C03083=1169.283,50.412,-48.994,-179.559,6.091,148.965
C03084=1169.288,50.162,-48.978,-179.562,6.091,148.965
C03085=1169.293,49.912,-48.962,-179.565,6.089,148.966
C03086=1169.298,49.663,-48.946,-179.567,6.089,148.966
C03087=1169.303,49.413,-48.930,-179.569,6.088,148.967
C03088=1169.308,49.164,-48.914,-179.573,6.086,148.967
C03089=1169.313,48.915,-48.899,-179.575,6.086,148.968
C03090=1169.318,48.665,-48.883,-179.577,6.085,148.969
C03091=1169.323,48.416,-48.867,-179.580,6.083,148.969
C03092=1169.328,48.167,-48.851,-179.583,6.083,148.970
C03093=1169.333,47.916,-48.835,-179.585,6.082,148.970
C03094=1169.338,47.667,-48.820,-179.588,6.081,148.971
C03095=1169.343,47.418,-48.805,-179.590,6.080,148.971
C03096=1169.348,47.168,-48.789,-179.593,6.079,148.972
C03097=1169.353,46.919,-48.773,-179.596,6.078,148.972
C03098=1169.358,46.670,-48.758,-179.598,6.077,148.973
C03099=1169.363,46.420,-48.742,-179.601,6.077,148.974
C03100=1169.368,46.171,-48.726,-179.604,6.075,148.974
C03101=1169.373,45.921,-48.711,-179.606,6.075,148.975
C03102=1169.378,45.672,-48.696,-179.609,6.074,148.975
C03103=1169.383,45.422,-48.680,-179.611,6.073,148.976
C03104=1169.388,45.173,-48.664,-179.614,6.072,148.976
C03105=1169.393,44.923,-48.648,-179.617,6.071,148.977
C03106=1169.398,44.674,-48.633,-179.619,6.070,148.978
C03107=1169.403,44.424,-48.617,-179.622,6.069,148.978
C03108=1169.408,44.175,-48.602,-179.624,6.068,148.979
C03109=1169.413,43.925,-48.587,-179.627,6.068,148.979
C03110=1169.418,43.676,-48.571,-179.630,6.066,148.980
C03111=1169.423,43.426,-48.555,-179.632,6.065,148.980
C03112=1169.428,43.177,-48.540,-179.635,6.065,148.981
C03113=1169.433,42.927,-48.525,-179.637,6.064,148.982
C03114=1169.439,42.678,-48.509,-179.640,6.063,148.982
C03115=1169.443,42.428,-48.494,-179.642,6.062,148.983
C03116=1169.448,42.179,-48.478,-179.645,6.061,148.983
C03117=1169.453,41.929,-48.463,-179.648,6.060,148.984
C03118=1169.458,41.680,-48.448,-179.650,6.059,148.984
C03119=1169.463,41.431,-48.432,-179.653,6.058,148.985
C03120=1169.468,41.181,-48.416,-179.655,6.058,148.986
C03121=1169.473,40.932,-48.401,-179.658,6.056,148.986
C03122=1169.478,40.682,-48.386,-179.661,6.056,148.987
C03123=1169.483,40.433,-48.371,-179.663,6.055,148.987
C03124=1169.488,40.184,-48.355,-179.666,6.054,148.988
C03125=1169.493,39.934,-48.339,-179.669,6.053,148.988
C03126=1169.498,39.684,-48.325,-179.671,6.052,148.989
C03127=1169.503,39.435,-48.309,-179.673,6.052,148.990
C03128=1169.508,39.186,-48.294,-179.676,6.050,148.990
C03129=1169.513,38.936,-48.279,-179.679,6.050,148.991
C03130=1169.519,38.687,-48.263,-179.681,6.049,148.991
C03131=1169.523,38.437,-48.248,-179.684,6.048,148.992
C03132=1169.529,38.187,-48.233,-179.686,6.047,148.992
C03133=1169.533,37.938,-48.218,-179.689,6.046,148.993
C03134=1169.539,37.688,-48.202,-179.692,6.046,148.994
C03135=1169.543,37.439,-48.187,-179.694,6.045,148.994
C03136=1169.549,37.190,-48.172,-179.697,6.043,148.995
C03137=1169.554,36.940,-48.157,-179.699,6.043,148.995
C03138=1169.559,36.691,-48.142,-179.702,6.042,148.996
C03139=1169.563,36.441,-48.126,-179.704,6.041,148.996
C03140=1169.568,36.192,-48.111,-179.707,6.040,148.997
C03141=1169.573,35.942,-48.096,-179.709,6.039,148.997
C03142=1169.579,35.693,-48.081,-179.712,6.039,148.998
C03143=1169.583,35.443,-48.066,-179.715,6.038,148.999
C03144=1169.589,35.193,-48.051,-179.717,6.036,148.999
C03145=1169.594,34.944,-48.036,-179.720,6.036,149.000
C03146=1169.599,34.695,-48.020,-179.722,6.035,149.000
C03147=1169.604,34.445,-48.006,-179.725,6.035,149.001
C03148=1169.609,34.196,-47.991,-179.728,6.033,149.001
C03149=1169.614,33.946,-47.975,-179.730,6.032,149.002
C03150=1169.618,33.696,-47.961,-179.733,6.032,149.003
C03151=1169.624,33.447,-47.945,-179.735,6.031,149.003
C03152=1169.629,33.198,-47.930,-179.738,6.030,149.004
C03153=1169.634,32.948,-47.915,-179.740,6.029,149.004
C03154=1169.639,32.699,-47.900,-179.743,6.028,149.005
C03155=1169.644,32.449,-47.885,-179.745,6.028,149.006
C03156=1169.649,32.200,-47.871,-179.748,6.027,149.006
C03157=1169.654,31.950,-47.856,-179.751,6.026,149.007
C03158=1169.660,31.700,-47.841,-179.753,6.025,149.007
C03159=1169.664,31.451,-47.826,-179.756,6.024,149.008
C03160=1169.669,31.202,-47.811,-179.758,6.024,149.008
C03161=1169.675,30.952,-47.796,-179.761,6.022,149.009
C03162=1169.679,30.703,-47.781,-179.763,6.021,149.010
C03163=1169.685,30.453,-47.766,-179.766,6.021,149.010
C03164=1169.690,30.204,-47.751,-179.769,6.021,149.011
C03165=1169.694,29.954,-47.737,-179.771,6.020,149.011
C03166=1169.700,29.705,-47.721,-179.774,6.018,149.012
C03167=1169.705,29.455,-47.707,-179.776,6.018,149.013
C03168=1169.709,29.206,-47.692,-179.779,6.017,149.013
C03169=1169.715,28.956,-47.677,-179.781,6.016,149.014
C03170=1169.720,28.707,-47.662,-179.784,6.016,149.014
C03171=1169.725,28.438,-47.646,-179.787,6.014,149.015
C03172=1169.731,28.169,-47.630,-179.790,6.014,149.016
C03173=1169.736,27.900,-47.614,-179.792,6.012,149.016
C03174=1169.741,27.632,-47.599,-179.795,6.012,149.017
C03175=1169.747,27.382,-47.584,-179.798,6.011,149.017
C03176=1169.752,27.132,-47.569,-179.800,6.010,149.018
C03177=1169.756,26.883,-47.554,-179.803,6.009,149.019
C03178=1169.761,26.633,-47.540,-179.805,6.008,149.019
C03179=1169.767,26.384,-47.525,-179.808,6.008,149.020
C03180=1169.772,26.134,-47.510,-179.811,6.007,149.020
C03181=1169.777,25.884,-47.496,-179.813,6.007,149.021
C03182=1169.781,25.635,-47.481,-179.815,6.006,149.022
C03183=1169.787,25.385,-47.466,-179.818,6.004,149.022
C03184=1169.792,25.135,-47.452,-179.821,6.004,149.023
C03185=1169.797,24.886,-47.437,-179.823,6.003,149.023
C03186=1169.801,24.637,-47.423,-179.826,6.003,149.024
C03187=1169.807,24.388,-47.409,-179.828,6.002,149.024
C03188=1169.812,24.138,-47.393,-179.831,6.000,149.025
C03189=1169.817,23.888,-47.379,-179.834,6.000,149.026
C03190=1169.822,23.639,-47.365,-179.836,5.999,149.026
C03191=1169.827,23.390,-47.350,-179.838,5.999,149.027
C03192=1169.832,23.140,-47.335,-179.841,5.998,149.027
C03193=1169.838,22.890,-47.320,-179.843,5.997,149.028
C03194=1169.843,22.640,-47.306,-179.846,5.996,149.029
C03195=1169.847,22.391,-47.291,-179.849,5.995,149.029
C03196=1169.852,22.141,-47.277,-179.851,5.995,149.030
C03197=1169.858,21.892,-47.263,-179.854,5.994,149.030
C03198=1169.863,21.643,-47.249,-179.856,5.993,149.031
C03199=1169.867,21.394,-47.234,-179.859,5.993,149.032
C03200=1169.873,21.144,-47.219,-179.862,5.991,149.032
C03201=1169.878,20.894,-47.205,-179.864,5.991,149.033
C03202=1169.883,20.644,-47.190,-179.867,5.990,149.033
C03203=1169.888,20.394,-47.176,-179.869,5.989,149.034
C03204=1169.893,20.145,-47.161,-179.872,5.989,149.034
C03205=1169.898,19.896,-47.147,-179.874,5.988,149.035
C03206=1169.903,19.647,-47.133,-179.876,5.988,149.036
C03207=1169.908,19.397,-47.119,-179.879,5.986,149.036
C03208=1169.913,19.147,-47.104,-179.882,5.986,149.037
C03209=1169.918,18.897,-47.090,-179.884,5.985,149.037
C03210=1169.923,18.648,-47.076,-179.887,5.984,149.038
C03211=1169.929,18.399,-47.060,-179.889,5.984,149.039
C03212=1169.934,18.149,-47.046,-179.891,5.983,149.039
C03213=1169.939,17.900,-47.032,-179.894,5.982,149.040
C03214=1169.944,17.650,-47.018,-179.897,5.981,149.040
C03215=1169.949,17.400,-47.003,-179.900,5.980,149.041
C03216=1169.954,17.151,-46.989,-179.902,5.980,149.042
C03217=1169.959,16.902,-46.975,-179.904,5.979,149.042
C03218=1169.964,16.652,-46.961,-179.907,5.978,149.043
C03219=1169.969,16.402,-46.947,-179.910,5.978,149.043
C03220=1169.974,16.152,-46.932,-179.912,5.977,149.044
C03221=1169.980,15.903,-46.918,-179.915,5.976,149.044
C03222=1169.985,15.654,-46.904,-179.917,5.975,149.045
C03223=1169.990,15.404,-46.890,-179.920,5.975,149.046
C03224=1169.995,15.154,-46.876,-179.922,5.974,149.046
C03225=1169.999,14.905,-46.861,-179.925,5.973,149.047
C03226=1170.005,14.656,-46.847,-179.927,5.973,149.047
C03227=1170.010,14.406,-46.833,-179.929,5.972,149.048
C03228=1170.015,14.156,-46.819,-179.932,5.971,149.049
C03229=1170.019,13.907,-46.805,-179.935,5.970,149.049
C03230=1170.025,13.658,-46.791,-179.938,5.969,149.050
C03231=1170.030,13.408,-46.777,-179.940,5.969,149.050
C03232=1170.035,13.158,-46.763,-179.942,5.968,149.051
C03233=1170.040,12.909,-46.748,-179.945,5.968,149.052
C03234=1170.045,12.660,-46.735,-179.948,5.967,149.052
C03235=1170.050,12.410,-46.720,-179.950,5.966,149.053
C03236=1170.055,12.160,-46.706,-179.952,5.966,149.053
C03237=1170.061,11.911,-46.693,-179.955,5.965,149.054
C03238=1170.066,11.661,-46.679,-179.958,5.964,149.055
C03239=1170.071,11.411,-46.664,-179.961,5.963,149.055
C03240=1170.076,11.161,-46.650,-179.963,5.962,149.056
C03241=1170.081,10.913,-46.637,-179.965,5.962,149.056
C03242=1170.086,10.663,-46.622,-179.968,5.961,149.057
C03243=1170.090,10.413,-46.608,-179.970,5.961,149.057
C03244=1170.096,10.164,-46.595,-179.973,5.960,149.058
C03245=1170.101,9.914,-46.581,-179.975,5.959,149.059
C03246=1170.106,9.664,-46.566,-179.978,5.959,149.059
C03247=1170.112,9.415,-46.552,-179.980,5.958,149.060
C03248=1170.116,9.166,-46.539,-179.982,5.958,149.060
C03249=1170.121,8.915,-46.525,-179.986,5.956,149.061
C03250=1170.126,8.666,-46.511,-179.988,5.955,149.062
C03251=1170.132,8.417,-46.497,-179.991,5.955,149.062
C03252=1170.137,8.167,-46.483,-179.993,5.955,149.063
C03253=1170.142,7.918,-46.470,-179.995,5.954,149.063
C03254=1170.147,7.668,-46.456,-179.998,5.953,149.064
C03255=1170.152,7.418,-46.442,180.000,5.952,149.065
C03256=1170.157,7.169,-46.428,179.997,5.952,149.065
C03257=1170.163,6.919,-46.414,179.995,5.951,149.066
C03258=1170.167,6.670,-46.400,179.992,5.951,149.066
C03259=1170.172,6.421,-46.386,179.990,5.950,149.067
C03260=1170.177,6.171,-46.372,179.988,5.949,149.068
C03261=1170.183,5.921,-46.359,179.984,5.948,149.068
C03262=1170.187,5.672,-46.345,179.982,5.948,149.069
C03263=1170.192,5.422,-46.331,179.979,5.947,149.069
C03264=1170.198,5.172,-46.318,179.977,5.946,149.070
C03265=1170.203,4.923,-46.304,179.974,5.946,149.071
C03266=1170.208,4.673,-46.291,179.972,5.945,149.071
C03267=1170.213,4.424,-46.277,179.969,5.944,149.072
C03268=1170.218,4.174,-46.262,179.967,5.944,149.072
C03269=1170.223,3.924,-46.249,179.965,5.943,149.073
C03270=1170.228,3.675,-46.236,179.962,5.943,149.074
C03271=1170.233,3.425,-46.221,179.960,5.942,149.074
C03272=1170.239,3.176,-46.208,179.957,5.941,149.075
C03273=1170.243,2.926,-46.194,179.955,5.941,149.075
C03274=1170.249,2.677,-46.181,179.952,5.940,149.076
C03275=1170.255,2.407,-46.166,179.949,5.939,149.077
C03276=1170.260,2.138,-46.151,179.946,5.938,149.077
C03277=1170.265,1.869,-46.137,179.944,5.938,149.078
C03278=1170.271,1.600,-46.122,179.941,5.937,149.079
C03279=1170.276,1.350,-46.109,179.939,5.937,149.079
C03280=1170.280,1.100,-46.095,179.936,5.936,149.080
C03281=1170.286,0.851,-46.082,179.934,5.935,149.080
C03282=1170.291,0.601,-46.067,179.931,5.935,149.081
C03283=1170.296,0.352,-46.055,179.929,5.934,149.082
C03284=1170.301,0.102,-46.041,179.927,5.934,149.082
C03285=1170.307,-0.148,-46.027,179.924,5.933,149.083
C03286=1170.311,-0.397,-46.014,179.921,5.932,149.083
C03287=1170.317,-0.647,-46.001,179.918,5.931,149.084
C03288=1170.321,-0.896,-45.987,179.916,5.931,149.085
C03289=1170.327,-1.146,-45.974,179.914,5.930,149.085
C03290=1170.332,-1.396,-45.960,179.911,5.929,149.086
C03291=1170.337,-1.645,-45.947,179.909,5.928,149.086
C03292=1170.343,-1.895,-45.933,179.906,5.928,149.087
C03293=1170.347,-2.144,-45.920,179.903,5.928,149.088
C03294=1170.353,-2.394,-45.906,179.901,5.927,149.088
C03295=1170.357,-2.643,-45.893,179.899,5.926,149.089
C03296=1170.363,-2.893,-45.879,179.896,5.925,149.089
C03297=1170.369,-3.143,-45.866,179.894,5.925,149.090
C03298=1170.373,-3.392,-45.853,179.891,5.925,149.091
C03299=1170.379,-3.642,-45.839,179.889,5.924,149.091
C03300=1170.383,-3.892,-45.826,179.886,5.923,149.092
C03301=1170.389,-4.141,-45.813,179.884,5.923,149.093
C03302=1170.393,-4.391,-45.800,179.882,5.922,149.093
C03303=1170.399,-4.641,-45.786,179.879,5.922,149.094
C03304=1170.403,-4.890,-45.773,179.877,5.921,149.094
C03305=1170.409,-5.140,-45.759,179.874,5.920,149.095
C03306=1170.414,-5.389,-45.747,179.871,5.920,149.096
C03307=1170.419,-5.639,-45.733,179.869,5.919,149.096
C03308=1170.424,-5.888,-45.720,179.867,5.918,149.097
C03309=1170.430,-6.138,-45.706,179.864,5.918,149.097
C03310=1170.434,-6.387,-45.693,179.862,5.917,149.098
C03311=1170.440,-6.637,-45.680,179.859,5.917,149.099
C03312=1170.445,-6.887,-45.667,179.857,5.916,149.099
C03313=1170.450,-7.136,-45.654,179.854,5.915,149.100
C03314=1170.455,-7.386,-45.640,179.852,5.915,149.100
C03315=1170.460,-7.635,-45.627,179.849,5.914,149.101
C03316=1170.465,-7.885,-45.614,179.847,5.914,149.102
C03317=1170.470,-8.135,-45.601,179.844,5.913,149.102
C03318=1170.476,-8.385,-45.588,179.842,5.912,149.103
C03319=1170.480,-8.634,-45.574,179.839,5.912,149.103
C03320=1170.486,-8.883,-45.562,179.837,5.911,149.104
C03321=1170.491,-9.133,-45.548,179.834,5.911,149.105
C03322=1170.496,-9.383,-45.536,179.832,5.910,149.105
C03323=1170.501,-9.633,-45.522,179.830,5.909,149.106
C03324=1170.506,-9.882,-45.509,179.827,5.909,149.106
C03325=1170.511,-10.131,-45.496,179.824,5.909,149.107
C03326=1170.516,-10.381,-45.483,179.822,5.908,149.108
C03327=1170.522,-10.631,-45.470,179.819,5.907,149.108
C03328=1170.527,-10.880,-45.457,179.817,5.906,149.109
C03329=1170.532,-11.130,-45.444,179.815,5.906,149.109
C03330=1170.537,-11.380,-45.431,179.812,5.906,149.110
C03331=1170.542,-11.630,-45.418,179.810,5.905,149.111
C03332=1170.547,-11.879,-45.404,179.807,5.904,149.111
C03333=1170.552,-12.128,-45.392,179.805,5.903,149.112
C03334=1170.557,-12.378,-45.379,179.802,5.903,149.112
C03335=1170.563,-12.628,-45.366,179.800,5.903,149.113
C03336=1170.568,-12.877,-45.353,179.797,5.902,149.114
C03337=1170.572,-13.127,-45.340,179.795,5.901,149.114
C03338=1170.578,-13.377,-45.327,179.792,5.901,149.115
C03339=1170.583,-13.626,-45.314,179.790,5.900,149.115
C03340=1170.588,-13.876,-45.301,179.788,5.900,149.116
C03341=1170.593,-14.125,-45.289,179.786,5.900,149.117
C03342=1170.599,-14.375,-45.275,179.783,5.899,149.117
C03343=1170.604,-14.624,-45.263,179.780,5.899,149.118
C03344=1170.608,-14.874,-45.250,179.778,5.898,149.118
C03345=1170.614,-15.124,-45.237,179.776,5.897,149.119
C03346=1170.619,-15.373,-45.224,179.773,5.897,149.120
C03347=1170.624,-15.623,-45.211,179.771,5.896,149.120
C03348=1170.629,-15.872,-45.199,179.768,5.896,149.121
C03349=1170.635,-16.122,-45.185,179.766,5.895,149.122
C03350=1170.639,-16.372,-45.172,179.763,5.894,149.122
C03351=1170.645,-16.621,-45.160,179.761,5.894,149.123
C03352=1170.650,-16.871,-45.147,179.758,5.893,149.123
C03353=1170.655,-17.120,-45.135,179.756,5.893,149.124
C03354=1170.660,-17.370,-45.121,179.753,5.892,149.125
C03355=1170.666,-17.620,-45.109,179.751,5.891,149.125
C03356=1170.671,-17.870,-45.097,179.748,5.891,149.126
C03357=1170.676,-18.119,-45.084,179.746,5.890,149.126
C03358=1170.681,-18.369,-45.070,179.743,5.890,149.127
C03359=1170.686,-18.619,-45.058,179.741,5.889,149.128
C03360=1170.691,-18.868,-45.045,179.739,5.889,149.128
C03361=1170.696,-19.117,-45.033,179.737,5.889,149.129
C03362=1170.701,-19.367,-45.020,179.734,5.888,149.130
C03363=1170.706,-19.617,-45.008,179.732,5.887,149.130
C03364=1170.712,-19.867,-44.995,179.729,5.887,149.131
C03365=1170.717,-20.116,-44.982,179.727,5.886,149.131
C03366=1170.722,-20.365,-44.969,179.724,5.886,149.132
C03367=1170.727,-20.615,-44.956,179.722,5.885,149.133
C03368=1170.732,-20.865,-44.944,179.719,5.885,149.133
C03369=1170.738,-21.115,-44.932,179.717,5.884,149.134
C03370=1170.743,-21.364,-44.919,179.714,5.884,149.135
C03371=1170.749,-21.614,-44.906,179.712,5.883,149.135
C03372=1170.753,-21.864,-44.893,179.709,5.882,149.136
C03373=1170.758,-22.114,-44.881,179.707,5.882,149.136
C03374=1170.764,-22.363,-44.869,179.705,5.882,149.137
C03375=1170.769,-22.612,-44.856,179.702,5.881,149.138
C03376=1170.774,-22.862,-44.843,179.700,5.881,149.138
C03377=1170.779,-23.112,-44.831,179.697,5.880,149.139
C03378=1170.784,-23.361,-44.819,179.695,5.880,149.139
C03379=1170.790,-23.631,-44.805,179.693,5.879,149.140
C03380=1170.795,-23.901,-44.792,179.690,5.879,149.141
C03381=1170.800,-24.171,-44.778,179.687,5.878,149.141
C03382=1170.807,-24.440,-44.764,179.685,5.878,149.142
C03383=1170.812,-24.690,-44.752,179.682,5.877,149.142
C03384=1170.817,-24.940,-44.739,179.680,5.876,149.143
C03385=1170.822,-25.190,-44.727,179.677,5.876,149.144
C03386=1170.827,-25.439,-44.715,179.675,5.875,149.144
C03387=1170.832,-25.689,-44.702,179.672,5.875,149.145
C03388=1170.838,-25.938,-44.690,179.670,5.874,149.146
C03389=1170.843,-26.188,-44.678,179.667,5.873,149.146
C03390=1170.848,-26.437,-44.665,179.665,5.873,149.147
C03391=1170.853,-26.687,-44.652,179.663,5.872,149.147
C03392=1170.858,-26.937,-44.640,179.661,5.873,149.148
C03393=1170.863,-27.187,-44.628,179.658,5.872,149.149
C03394=1170.869,-27.437,-44.616,179.656,5.871,149.149
C03395=1170.874,-27.686,-44.603,179.653,5.871,149.150
C03396=1170.879,-27.935,-44.591,179.650,5.870,149.151
C03397=1170.884,-28.185,-44.579,179.648,5.870,149.151
C03398=1170.889,-28.434,-44.566,179.646,5.869,149.152
C03399=1170.894,-28.685,-44.554,179.643,5.868,149.152
C03400=1170.899,-28.934,-44.541,179.641,5.868,149.153
C03401=1170.904,-29.184,-44.530,179.639,5.868,149.154
C03402=1170.909,-29.433,-44.517,179.636,5.867,149.154
C03403=1170.915,-29.683,-44.505,179.634,5.867,149.155
C03404=1170.920,-29.933,-44.493,179.631,5.867,149.155
C03405=1170.925,-30.182,-44.480,179.629,5.866,149.156
C03406=1170.930,-30.432,-44.468,179.626,5.865,149.157
C03407=1170.935,-30.681,-44.456,179.624,5.865,149.157
C03408=1170.941,-30.931,-44.444,179.621,5.864,149.158
C03409=1170.946,-31.181,-44.432,179.619,5.864,149.159
C03410=1170.951,-31.430,-44.419,179.617,5.864,149.159
C03411=1170.957,-31.680,-44.407,179.615,5.863,149.160
C03412=1170.961,-31.929,-44.395,179.612,5.862,149.160
C03413=1170.967,-32.179,-44.384,179.610,5.862,149.161
C03414=1170.972,-32.429,-44.371,179.607,5.862,149.162
C03415=1170.977,-32.679,-44.359,179.605,5.861,149.162
C03416=1170.982,-32.929,-44.346,179.602,5.860,149.163
C03417=1170.987,-33.178,-44.334,179.600,5.861,149.163
C03418=1170.993,-33.428,-44.322,179.598,5.860,149.164
C03419=1170.998,-33.678,-44.310,179.595,5.859,149.165
C03420=1171.002,-33.927,-44.298,179.593,5.859,149.165
C03421=1171.008,-34.177,-44.286,179.590,5.858,149.166
C03422=1171.013,-34.427,-44.274,179.588,5.858,149.166
C03423=1171.018,-34.677,-44.262,179.586,5.857,149.167
C03424=1171.024,-34.926,-44.250,179.584,5.857,149.168
C03425=1171.029,-35.176,-44.238,179.581,5.856,149.168
C03426=1171.034,-35.425,-44.226,179.579,5.856,149.169
C03427=1171.039,-35.675,-44.214,179.576,5.856,149.170
C03428=1171.044,-35.925,-44.202,179.574,5.855,149.170
C03429=1171.050,-36.175,-44.190,179.571,5.854,149.171
C03430=1171.055,-36.424,-44.177,179.568,5.854,149.171
C03431=1171.059,-36.674,-44.166,179.567,5.854,149.172
C03432=1171.065,-36.923,-44.154,179.564,5.853,149.173
C03433=1171.071,-37.172,-44.142,179.562,5.853,149.173
C03434=1171.076,-37.422,-44.130,179.559,5.852,149.174
C03435=1171.081,-37.672,-44.119,179.557,5.852,149.174
C03436=1171.086,-37.921,-44.106,179.555,5.851,149.175
C03437=1171.091,-38.171,-44.094,179.552,5.851,149.176
C03438=1171.097,-38.421,-44.082,179.550,5.851,149.176
C03439=1171.101,-38.670,-44.071,179.548,5.850,149.177
C03440=1171.106,-38.920,-44.059,179.545,5.850,149.177
C03441=1171.112,-39.170,-44.047,179.543,5.849,149.178
C03442=1171.117,-39.420,-44.035,179.540,5.848,149.179
C03443=1171.122,-39.669,-44.023,179.538,5.849,149.179
C03444=1171.127,-39.919,-44.012,179.536,5.848,149.180
C03445=1171.133,-40.169,-43.999,179.533,5.848,149.181
C03446=1171.138,-40.418,-43.987,179.531,5.847,149.181
C03447=1171.143,-40.668,-43.976,179.528,5.846,149.182
C03448=1171.149,-40.917,-43.964,179.526,5.846,149.182
C03449=1171.154,-41.167,-43.952,179.524,5.846,149.183
C03450=1171.159,-41.416,-43.940,179.521,5.846,149.184
C03451=1171.164,-41.666,-43.929,179.519,5.845,149.184
C03452=1171.169,-41.916,-43.917,179.517,5.844,149.185
C03453=1171.174,-42.166,-43.905,179.514,5.844,149.185
C03454=1171.180,-42.416,-43.893,179.512,5.843,149.186
C03455=1171.185,-42.666,-43.882,179.510,5.843,149.187
C03456=1171.190,-42.915,-43.870,179.507,5.843,149.187
C03457=1171.195,-43.165,-43.858,179.505,5.842,149.188
C03458=1171.200,-43.414,-43.847,179.502,5.842,149.189
C03459=1171.206,-43.663,-43.835,179.500,5.841,149.189
C03460=1171.211,-43.913,-43.823,179.498,5.841,149.190
C03461=1171.216,-44.163,-43.812,179.496,5.841,149.190
C03462=1171.221,-44.413,-43.800,179.493,5.840,149.191
C03463=1171.226,-44.663,-43.788,179.490,5.840,149.192
C03464=1171.231,-44.913,-43.777,179.488,5.839,149.192
C03465=1171.237,-45.162,-43.765,179.486,5.839,149.193
C03466=1171.242,-45.411,-43.754,179.484,5.838,149.193
C03467=1171.247,-45.661,-43.742,179.481,5.838,149.194
C03468=1171.252,-45.911,-43.731,179.479,5.838,149.195
C03469=1171.257,-46.161,-43.719,179.476,5.837,149.195
C03470=1171.263,-46.411,-43.707,179.474,5.837,149.196
C03471=1171.268,-46.660,-43.696,179.472,5.836,149.196
C03472=1171.274,-46.910,-43.684,179.470,5.836,149.197
C03473=1171.278,-47.159,-43.673,179.467,5.835,149.198
C03474=1171.284,-47.409,-43.661,179.465,5.835,149.198
C03475=1171.288,-47.659,-43.650,179.463,5.835,149.199
C03476=1171.294,-47.909,-43.638,179.460,5.834,149.199
C03477=1171.299,-48.158,-43.627,179.458,5.834,149.200
C03478=1171.305,-48.408,-43.615,179.455,5.833,149.201
C03479=1171.310,-48.658,-43.603,179.453,5.833,149.201
C03480=1171.315,-48.907,-43.592,179.451,5.833,149.202
C03481=1171.320,-49.157,-43.580,179.449,5.832,149.202
C03482=1171.325,-49.406,-43.569,179.446,5.832,149.203
C03483=1171.331,-49.677,-43.557,179.443,5.831,149.204
C03484=1171.336,-49.947,-43.544,179.441,5.831,149.204
C03485=1171.343,-50.218,-43.532,179.438,5.830,149.205
C03486=1171.348,-50.488,-43.519,179.436,5.830,149.206
C03487=1171.353,-50.738,-43.508,179.434,5.830,149.206
C03488=1171.359,-50.988,-43.497,179.432,5.829,149.207
C03489=1171.364,-51.237,-43.485,179.429,5.829,149.208
C03490=1171.369,-51.487,-43.474,179.426,5.828,149.208
C03491=1171.374,-51.737,-43.462,179.424,5.828,149.209
C03492=1171.380,-51.986,-43.451,179.422,5.828,149.209
C03493=1171.384,-52.236,-43.439,179.420,5.827,149.210
C03494=1171.389,-52.486,-43.429,179.417,5.827,149.211
C03495=1171.395,-52.736,-43.417,179.414,5.826,149.211
C03496=1171.400,-52.985,-43.406,179.413,5.826,149.212
C03497=1171.406,-53.235,-43.394,179.410,5.826,149.212
C03498=1171.410,-53.484,-43.383,179.408,5.825,149.213
C03499=1171.416,-53.734,-43.371,179.405,5.825,149.214
C03500=1171.421,-53.984,-43.361,179.403,5.824,149.214
C03501=1171.426,-54.233,-43.350,179.401,5.824,149.215
C03502=1171.431,-54.483,-43.338,179.398,5.824,149.216
C03503=1171.436,-54.733,-43.326,179.396,5.823,149.216
C03504=1171.442,-54.982,-43.316,179.393,5.823,149.217
C03505=1171.447,-55.232,-43.304,179.391,5.823,149.217
C03506=1171.452,-55.482,-43.293,179.389,5.822,149.218
C03507=1171.458,-55.731,-43.281,179.387,5.822,149.219
C03508=1171.463,-55.981,-43.271,179.384,5.821,149.219
C03509=1171.468,-56.231,-43.260,179.382,5.821,149.220
C03510=1171.473,-56.481,-43.248,179.380,5.821,149.220
C03511=1171.478,-56.730,-43.237,179.377,5.820,149.221
C03512=1171.483,-56.980,-43.226,179.375,5.820,149.222
C03513=1171.489,-57.230,-43.214,179.373,5.820,149.222
C03514=1171.494,-57.479,-43.203,179.371,5.819,149.223
C03515=1171.499,-57.729,-43.193,179.368,5.819,149.223
C03516=1171.504,-57.979,-43.181,179.366,5.818,149.224
C03517=1171.510,-58.228,-43.170,179.364,5.819,149.225
C03518=1171.515,-58.478,-43.159,179.361,5.818,149.225
C03519=1171.520,-58.728,-43.148,179.359,5.817,149.226
C03520=1171.525,-58.977,-43.137,179.357,5.817,149.226
C03521=1171.530,-59.228,-43.126,179.354,5.817,149.227
C03522=1171.535,-59.477,-43.115,179.352,5.816,149.228
C03523=1171.541,-59.727,-43.104,179.350,5.816,149.228
C03524=1171.546,-59.977,-43.093,179.347,5.815,149.229
C03525=1171.551,-60.226,-43.081,179.345,5.815,149.229
C03526=1171.556,-60.476,-43.071,179.343,5.815,149.230
C03527=1171.562,-60.726,-43.059,179.341,5.814,149.231
C03528=1171.567,-60.975,-43.049,179.338,5.814,149.231
C03529=1171.572,-61.225,-43.038,179.336,5.814,149.232
C03530=1171.577,-61.475,-43.027,179.334,5.813,149.233
C03531=1171.583,-61.724,-43.016,179.331,5.813,149.233
C03532=1171.588,-61.974,-43.004,179.329,5.813,149.234
C03533=1171.593,-62.224,-42.994,179.327,5.812,149.234
C03534=1171.598,-62.473,-42.983,179.324,5.812,149.235
C03535=1171.604,-62.724,-42.972,179.322,5.811,149.236
C03536=1171.609,-62.973,-42.961,179.320,5.811,149.236
C03537=1171.614,-63.223,-42.950,179.318,5.811,149.237
C03538=1171.619,-63.473,-42.939,179.315,5.810,149.238
C03539=1171.624,-63.722,-42.929,179.313,5.810,149.238
C03540=1171.630,-63.972,-42.917,179.311,5.810,149.239
C03541=1171.636,-64.222,-42.907,179.308,5.809,149.239
C03542=1171.640,-64.471,-42.895,179.306,5.809,149.240
C03543=1171.646,-64.721,-42.885,179.304,5.809,149.240
C03544=1171.650,-64.970,-42.874,179.301,5.808,149.241
C03545=1171.656,-65.221,-42.863,179.299,5.808,149.242
C03546=1171.662,-65.470,-42.852,179.297,5.808,149.242
C03547=1171.667,-65.720,-42.841,179.295,5.808,149.243
C03548=1171.672,-65.969,-42.830,179.292,5.807,149.243
C03549=1171.677,-66.219,-42.820,179.290,5.806,149.244
C03550=1171.682,-66.469,-42.809,179.288,5.806,149.245
C03551=1171.687,-66.718,-42.798,179.285,5.806,149.245
C03552=1171.693,-66.968,-42.787,179.283,5.806,149.246
C03553=1171.698,-67.218,-42.776,179.281,5.806,149.247
C03554=1171.704,-67.467,-42.766,179.279,5.805,149.247
C03555=1171.708,-67.717,-42.755,179.276,5.804,149.248
C03556=1171.713,-67.967,-42.744,179.274,5.804,149.248
C03557=1171.719,-68.217,-42.734,179.272,5.804,149.249
C03558=1171.724,-68.466,-42.723,179.269,5.804,149.250
C03559=1171.729,-68.716,-42.712,179.267,5.803,149.250
C03560=1171.735,-68.967,-42.701,179.265,5.803,149.251
C03561=1171.740,-69.216,-42.690,179.262,5.803,149.252
C03562=1171.745,-69.466,-42.680,179.260,5.802,149.252
C03563=1171.751,-69.715,-42.669,179.258,5.802,149.253
C03564=1171.756,-69.965,-42.658,179.256,5.802,149.253
C03565=1171.761,-70.214,-42.648,179.253,5.801,149.254
C03566=1171.766,-70.465,-42.637,179.251,5.800,149.254
C03567=1171.772,-70.714,-42.626,179.249,5.801,149.255
C03568=1171.777,-70.964,-42.616,179.247,5.800,149.256
C03569=1171.782,-71.213,-42.606,179.244,5.800,149.256
C03570=1171.787,-71.464,-42.595,179.242,5.800,149.257
C03571=1171.792,-71.713,-42.584,179.240,5.799,149.257
C03572=1171.798,-71.962,-42.574,179.237,5.799,149.258
C03573=1171.803,-72.212,-42.563,179.236,5.799,149.259
C03574=1171.808,-72.461,-42.552,179.233,5.798,149.259
C03575=1171.813,-72.712,-42.542,179.231,5.798,149.260
C03576=1171.819,-72.961,-42.532,179.229,5.798,149.261
C03577=1171.824,-73.211,-42.521,179.227,5.797,149.261
C03578=1171.830,-73.461,-42.510,179.224,5.797,149.262
C03579=1171.835,-73.711,-42.499,179.222,5.797,149.262
C03580=1171.841,-73.960,-42.489,179.220,5.796,149.263
C03581=1171.846,-74.211,-42.478,179.217,5.796,149.264
C03582=1171.850,-74.460,-42.469,179.215,5.796,149.264
C03583=1171.856,-74.709,-42.458,179.213,5.796,149.265
C03584=1171.861,-74.959,-42.447,179.210,5.795,149.265
C03585=1171.866,-75.209,-42.437,179.208,5.795,149.266
C03586=1171.871,-75.459,-42.426,179.206,5.794,149.266
C03587=1171.878,-75.730,-42.415,179.204,5.794,149.267
C03588=1171.884,-76.001,-42.404,179.201,5.794,149.268
C03589=1171.889,-76.272,-42.392,179.199,5.793,149.268
C03590=1171.895,-76.543,-42.381,179.197,5.793,149.269
C03591=1171.900,-76.793,-42.370,179.194,5.793,149.270
C03592=1171.906,-77.043,-42.360,179.192,5.792,149.270
C03593=1171.911,-77.292,-42.350,179.190,5.792,149.271
C03594=1171.916,-77.542,-42.340,179.187,5.792,149.271
C03595=1171.921,-77.792,-42.330,179.185,5.791,149.272
C03596=1171.926,-78.041,-42.318,179.183,5.791,149.273
C03597=1171.931,-78.291,-42.308,179.181,5.791,149.273
C03598=1171.937,-78.540,-42.298,179.178,5.790,149.274
C03599=1171.942,-78.791,-42.287,179.176,5.790,149.275
C03600=1171.948,-79.040,-42.277,179.174,5.790,149.275
C03601=1171.953,-79.290,-42.267,179.171,5.789,149.276
C03602=1171.958,-79.540,-42.256,179.169,5.790,149.276
C03603=1171.964,-79.790,-42.246,179.167,5.789,149.277
C03604=1171.968,-80.039,-42.236,179.164,5.788,149.278
C03605=1171.974,-80.289,-42.226,179.163,5.788,149.278
C03606=1171.979,-80.539,-42.216,179.160,5.788,149.279
C03607=1171.984,-80.789,-42.205,179.158,5.787,149.279
C03608=1171.990,-81.038,-42.195,179.156,5.788,149.280
C03609=1171.995,-81.288,-42.185,179.154,5.787,149.281
C03610=1172.000,-81.538,-42.174,179.151,5.787,149.281
C03611=1172.005,-81.787,-42.165,179.149,5.787,149.282
C03612=1172.011,-82.037,-42.154,179.147,5.786,149.282
C03613=1172.016,-82.287,-42.144,179.145,5.786,149.283
C03614=1172.022,-82.537,-42.134,179.143,5.786,149.284
C03615=1172.027,-82.786,-42.123,179.140,5.785,149.284
C03616=1172.031,-83.036,-42.113,179.138,5.785,149.285
C03617=1172.037,-83.286,-42.103,179.136,5.785,149.285
C03618=1172.043,-83.535,-42.093,179.133,5.784,149.286
C03619=1172.048,-83.785,-42.082,179.132,5.784,149.286
C03620=1172.053,-84.035,-42.072,179.129,5.784,149.287
C03621=1172.058,-84.284,-42.063,179.127,5.783,149.288
C03622=1172.063,-84.535,-42.052,179.125,5.783,149.288
C03623=1172.069,-84.784,-42.042,179.123,5.783,149.289
C03624=1172.075,-85.034,-42.032,179.121,5.783,149.290
C03625=1172.079,-85.283,-42.023,179.118,5.782,149.290
C03626=1172.084,-85.534,-42.012,179.116,5.782,149.291
C03627=1172.090,-85.783,-42.002,179.114,5.782,149.291
C03628=1172.096,-86.033,-41.992,179.111,5.781,149.292
C03629=1172.100,-86.283,-41.982,179.109,5.781,149.293
C03630=1172.105,-86.532,-41.971,179.107,5.781,149.293
C03631=1172.111,-86.782,-41.961,179.105,5.781,149.294
C03632=1172.117,-87.032,-41.952,179.103,5.781,149.294
C03633=1172.121,-87.282,-41.942,179.100,5.780,149.295
C03634=1172.127,-87.531,-41.932,179.098,5.780,149.296
C03635=1172.132,-87.781,-41.921,179.096,5.780,149.296
C03636=1172.138,-88.031,-41.911,179.094,5.779,149.297
C03637=1172.142,-88.280,-41.901,179.091,5.779,149.297
C03638=1172.148,-88.531,-41.892,179.090,5.779,149.298
C03639=1172.154,-88.780,-41.882,179.087,5.778,149.299
C03640=1172.159,-89.029,-41.872,179.085,5.778,149.299
C03641=1172.164,-89.280,-41.861,179.083,5.778,149.300
C03642=1172.169,-89.529,-41.851,179.080,5.777,149.300
C03643=1172.174,-89.779,-41.842,179.079,5.777,149.301
C03644=1172.180,-90.029,-41.832,179.076,5.777,149.301
C03645=1172.185,-90.279,-41.821,179.075,5.777,149.302
C03646=1172.190,-90.528,-41.812,179.072,5.776,149.303
C03647=1172.196,-90.778,-41.802,179.070,5.776,149.303
C03648=1172.201,-91.028,-41.792,179.068,5.776,149.304
C03649=1172.206,-91.278,-41.782,179.065,5.775,149.304
